KUKA KRL program: EPS_2_251349_CBMH112_A_20251001124303.src

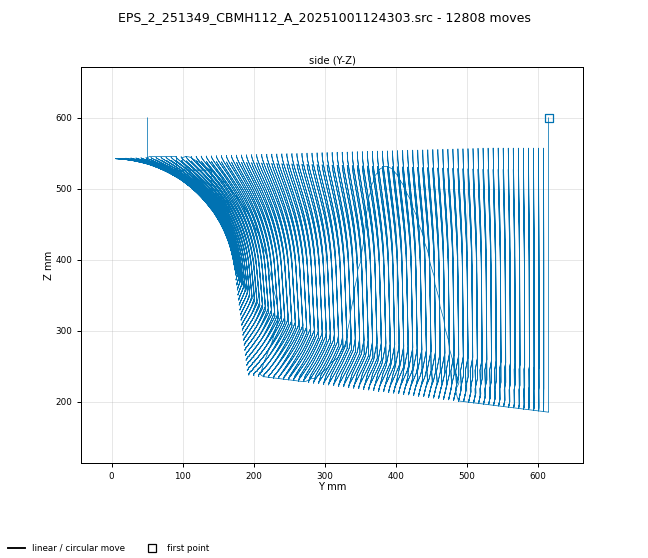
[picture p0: tool path of EPS_2_251349_CBMH112_A_20251001124303.src, 12808 of 12810 moves have a stored position in this frame; points joined in program order, loops and branches not executed]
&ACCESS RVP
&REL 4
&COMMENT QRS 19112012
&PARAM EDITMASK = *
DEF PART()
EXT BAS (BAS_COMMAND :IN,REAL :IN )
INT I
BAS (#INITMOV,0 )

;KUKA QRS Post kuka4.cps  Date:22-06-2017 !

File_ID=2860

QRS_PRE_INIT()

;Init var - Until changes are made in qrs_pre_init
Outlet_Square_prg=0
Inlet_1_Square_prg=0
Inlet_2_Square_prg=0
Inlet_3_Square_prg=0
Inlet_4_Square_prg=0
Inlet_5_Square_prg=0

Outlet_1={X 0.000, Y 529.100, Z 408.000, B 0.000, E1 0.000 }
Inlet_1={X 0.000, Y 531.280, Z 378.000, B 0.000, E1 180.000 }
Outlet_1_type=299
Inlet_1_type=299
;QRS#1=Sidecore dimensions
;QRS#2=300-12" PVC SDR 35
;QRS#3=300-12" PVC SDR 35
;QRS#4=
;QRS#5=
;QRS#6=
;QRS#7=
;QRS#8=
;QRS#9=16M PSX
;QRS#10=16M PSX
;QRS#11=
;QRS#12=
;QRS#13=
;QRS#14=
;QRS#15=
;QRS#16=1220x127x838 2,75'
;QRS#17=EPS Height
;QRS#18=557,5
;QRS#19=*
;QRS#20= UPDATED VERSION 22-06-2017
;QRS#21=*
Outlet_Square=0150
Inlet_1_Square=0150
Inlet_2_Square=0
Inlet_3_Square=0
Inlet_4_Square=0
Inlet_5_Square=0
Mill_Square=1
Outlet_Square_Prg=206
Inlet_1_Square_prg=206

QRS_INIT()

$ADVANCE=5

; T1
PTP {E1 173.597,E2 173.597}
PTP {X 0,Y 615.502,A -85,B 0,C 180,E1 173.597,E2 173.597,E3 0,E4 0,E5 0,E6 0}
QRS_SPEED_INIT()
LIN {X 0,Y 615.502,Z 600,A -85,B 0,C 180,E1 173.597,E2 173.597,E3 0,E4 0,E5 0,E6 0} C_VEL
LIN {X 0,Y 615.502,Z 195.488,A -85,B 0,C 180,E1 173.597,E2 173.597} C_VEL
LIN {X 0,Y 615.502,Z 187.309,A -85,B 0,C 180,E1 173.597,E2 173.597} C_VEL
LIN {X 0,Y 615.487,Z 185.309,A -85,B 0,C 180,E1 173.411,E2 173.411} C_VEL
LIN {X 0,Y 615.496,Z 185.324,A -85,B 0,C 180,E1 170.801,E2 170.801} C_VEL
LIN {X 0,Y 615.474,Z 185.313,A -85,B 0,C 180,E1 168.139,E2 168.139} C_VEL
LIN {X 0,Y 615.483,Z 185.311,A -85,B 0,C 180,E1 165.451,E2 165.451} C_VEL
LIN {X 0,Y 615.488,Z 185.323,A -85,B 0,C 180,E1 162.729,E2 162.729} C_VEL
LIN {X 0,Y 615.489,Z 185.307,A -85,B 0,C 180,E1 159.967,E2 159.967} C_VEL
LIN {X 0,Y 615.483,Z 185.321,A -85,B 0,C 180,E1 157.155,E2 157.155} C_VEL
LIN {X 0,Y 615.476,Z 185.315,A -85,B 0,C 180,E1 154.431,E2 154.431} C_VEL
LIN {X 0,Y 615.483,Z 185.309,A -85,B 0,C 180,E1 152.085,E2 152.085} C_VEL
LIN {X 0,Y 615.488,Z 185.308,A -85,B 0,C 180,E1 149.84,E2 149.84} C_VEL
LIN {X 0,Y 615.477,Z 185.315,A -85,B 0,C 180,E1 147.542,E2 147.542} C_VEL
LIN {X 0,Y 615.491,Z 185.323,A -85,B 0,C 180,E1 145.185,E2 145.185} C_VEL
LIN {X 0,Y 615.479,Z 185.318,A -85,B 0,C 180,E1 142.757,E2 142.757} C_VEL
LIN {X 0,Y 615.483,Z 185.31,A -85,B 0,C 180,E1 139.91,E2 139.91} C_VEL
LIN {X 0,Y 615.477,Z 185.316,A -85,B 0,C 180,E1 137.646,E2 137.646} C_VEL
LIN {X 0,Y 615.482,Z 185.319,A -85,B 0,C 180,E1 134.931,E2 134.931} C_VEL
LIN {X 0,Y 615.484,Z 185.309,A -85,B 0,C 180,E1 132.08,E2 132.08} C_VEL
LIN {X 0,Y 615.476,Z 185.316,A -85,B 0,C 180,E1 129.75,E2 129.75} C_VEL
LIN {X 0,Y 615.48,Z 185.317,A -85,B 0,C 180,E1 126.936,E2 126.936} C_VEL
LIN {X 0,Y 615.483,Z 185.311,A -85,B 0,C 180,E1 124.7,E2 124.7} C_VEL
LIN {X 0,Y 615.489,Z 185.307,A -85,B 0,C 180,E1 122.331,E2 122.331} C_VEL
LIN {X 0,Y 615.491,Z 185.326,A -85,B 0,C 180,E1 119.405,E2 119.405} C_VEL
LIN {X 0,Y 615.485,Z 185.308,A -85,B 0,C 180,E1 116.444,E2 116.444} C_VEL
LIN {X 0,Y 615.485,Z 185.327,A -85,B 0,C 180,E1 113.556,E2 113.556} C_VEL
LIN {X 0,Y 615.476,Z 185.338,A -85,B 0,C 180,E1 112.266,E2 112.266} C_VEL
LIN {X 0,Y 615.46,Z 205.213,A -85,B 0,C 180,E1 109.685,E2 109.685} C_VEL
LIN {X 0,Y 615.464,Z 216.791,A -85,B 0,C 180,E1 108.2,E2 108.2} C_VEL
LIN {X 0,Y 615.491,Z 381.255,A -85,B 0,C 180,E1 106.201,E2 106.201} C_VEL
LIN {X 0,Y 615.489,Z 395.834,A -85,B 0,C 180,E1 105.905,E2 105.905} C_VEL
LIN {X 0,Y 615.477,Z 410.429,A -85,B 0,C 180,E1 105.48,E2 105.48} C_VEL
LIN {X 0,Y 615.492,Z 423.747,A -85,B 0,C 180,E1 104.971,E2 104.971} C_VEL
LIN {X 0,Y 615.483,Z 437.385,A -85,B 0,C 180,E1 104.319,E2 104.319} C_VEL
LIN {X 0,Y 615.5,Z 450.671,A -85,B 0,C 180,E1 103.537,E2 103.537} C_VEL
LIN {X 0,Y 615.497,Z 462.521,A -85,B 0,C 180,E1 102.697,E2 102.697} C_VEL
LIN {X 0,Y 615.497,Z 474.363,A -85,B 0,C 180,E1 101.693,E2 101.693} C_VEL
LIN {X 0,Y 615.495,Z 484.168,A -85,B 0,C 180,E1 100.708,E2 100.708} C_VEL
LIN {X 0,Y 615.495,Z 494.014,A -85,B 0,C 180,E1 99.53,E2 99.53} C_VEL
LIN {X 0,Y 615.496,Z 502.104,A -85,B 0,C 180,E1 98.371,E2 98.371} C_VEL
LIN {X 0,Y 615.491,Z 508.784,A -85,B 0,C 180,E1 97.215,E2 97.215} C_VEL
LIN {X 0,Y 615.499,Z 514.949,A -85,B 0,C 180,E1 95.898,E2 95.898} C_VEL
LIN {X 0,Y 615.489,Z 519.717,A -85,B 0,C 180,E1 94.584,E2 94.584} C_VEL
LIN {X 0,Y 615.491,Z 523.221,A -85,B 0,C 180,E1 93.273,E2 93.273} C_VEL
LIN {X 0,Y 615.5,Z 525.54,A -85,B 0,C 180,E1 91.963,E2 91.963} C_VEL
LIN {X 0,Y 615.491,Z 526.728,A -85,B 0,C 180,E1 90.654,E2 90.654} C_VEL
LIN {X 0,Y 615.492,Z 526.751,A -85,B 0,C 180,E1 89.346,E2 89.346} C_VEL
LIN {X 0,Y 615.5,Z 525.646,A -85,B 0,C 180,E1 88.037,E2 88.037} C_VEL
LIN {X 0,Y 615.494,Z 523.416,A -85,B 0,C 180,E1 86.727,E2 86.727} C_VEL
LIN {X 0,Y 615.49,Z 520.005,A -85,B 0,C 180,E1 85.416,E2 85.416} C_VEL
LIN {X 0,Y 615.499,Z 515.336,A -85,B 0,C 180,E1 84.102,E2 84.102} C_VEL
LIN {X 0,Y 615.49,Z 509.273,A -85,B 0,C 180,E1 82.785,E2 82.785} C_VEL
LIN {X 0,Y 615.493,Z 501.634,A -85,B 0,C 180,E1 81.464,E2 81.464} C_VEL
LIN {X 0,Y 615.496,Z 493.451,A -85,B 0,C 180,E1 80.304,E2 80.304} C_VEL
LIN {X 0,Y 615.495,Z 483.338,A -85,B 0,C 180,E1 79.109,E2 79.109} C_VEL
LIN {X 0,Y 615.497,Z 471.686,A -85,B 0,C 180,E1 77.973,E2 77.973} C_VEL
LIN {X 0,Y 615.498,Z 460.416,A -85,B 0,C 180,E1 77.051,E2 77.051} C_VEL
LIN {X 0,Y 615.498,Z 448.178,A -85,B 0,C 180,E1 76.211,E2 76.211} C_VEL
LIN {X 0,Y 615.484,Z 434.781,A -85,B 0,C 180,E1 75.451,E2 75.451} C_VEL
LIN {X 0,Y 615.488,Z 419.868,A -85,B 0,C 180,E1 74.774,E2 74.774} C_VEL
LIN {X 0,Y 615.476,Z 405.395,A -85,B 0,C 180,E1 74.265,E2 74.265} C_VEL
LIN {X 0,Y 615.492,Z 389.76,A -85,B 0,C 180,E1 73.865,E2 73.865} C_VEL
LIN {X 0,Y 615.492,Z 374.754,A -85,B 0,C 180,E1 73.618,E2 73.618} C_VEL
LIN {X 0,Y 615.471,Z 216.859,A -85,B 0,C 180,E1 71.719,E2 71.719} C_VEL
LIN {X 0,Y 615.478,Z 195.117,A -85,B 0,C 180,E1 68.919,E2 68.919} C_VEL
LIN {X 0,Y 615.483,Z 185.31,A -85,B 0,C 180,E1 67.625,E2 67.625} C_VEL
LIN {X 0,Y 615.478,Z 185.313,A -85,B 0,C 180,E1 65.008,E2 65.008} C_VEL
LIN {X 0,Y 615.476,Z 185.318,A -85,B 0,C 180,E1 62.823,E2 62.823} C_VEL
LIN {X 0,Y 615.482,Z 185.319,A -85,B 0,C 180,E1 60.207,E2 60.207} C_VEL
LIN {X 0,Y 615.493,Z 185.306,A -85,B 0,C 180,E1 57.544,E2 57.544} C_VEL
LIN {X 0,Y 615.478,Z 185.312,A -85,B 0,C 180,E1 55.185,E2 55.185} C_VEL
LIN {X 0,Y 615.486,Z 185.322,A -85,B 0,C 180,E1 52.759,E2 52.759} C_VEL
LIN {X 0,Y 615.482,Z 185.31,A -85,B 0,C 180,E1 49.912,E2 49.912} C_VEL
LIN {X 0,Y 615.495,Z 185.306,A -85,B 0,C 180,E1 47.649,E2 47.649} C_VEL
LIN {X 0,Y 615.479,Z 185.322,A -85,B 0,C 180,E1 44.932,E2 44.932} C_VEL
LIN {X 0,Y 615.483,Z 185.311,A -85,B 0,C 180,E1 42.081,E2 42.081} C_VEL
LIN {X 0,Y 615.489,Z 185.307,A -85,B 0,C 180,E1 39.75,E2 39.75} C_VEL
LIN {X 0,Y 615.482,Z 185.325,A -85,B 0,C 180,E1 36.938,E2 36.938} C_VEL
LIN {X 0,Y 615.488,Z 185.308,A -85,B 0,C 180,E1 34.022,E2 34.022} C_VEL
LIN {X 0,Y 615.479,Z 185.323,A -85,B 0,C 180,E1 31.087,E2 31.087} C_VEL
LIN {X 0,Y 615.481,Z 185.314,A -85,B 0,C 180,E1 28.452,E2 28.452} C_VEL
LIN {X 0,Y 615.476,Z 185.311,A -85,B 0,C 180,E1 25.716,E2 25.716} C_VEL
LIN {X 0,Y 615.473,Z 185.315,A -85,B 0,C 180,E1 23.557,E2 23.557} C_VEL
LIN {X 0,Y 615.475,Z 185.318,A -85,B 0,C 180,E1 21.432,E2 21.432} C_VEL
LIN {X 0,Y 615.482,Z 185.314,A -85,B 0,C 180,E1 18.607,E2 18.607} C_VEL
LIN {X 0,Y 615.477,Z 185.311,A -85,B 0,C 180,E1 15.906,E2 15.906} C_VEL
LIN {X 0,Y 615.492,Z 185.325,A -85,B 0,C 180,E1 13.201,E2 13.201} C_VEL
LIN {X 0,Y 615.488,Z 185.31,A -85,B 0,C 180,E1 10.527,E2 10.527} C_VEL
LIN {X 0,Y 615.471,Z 185.314,A -85,B 0,C 180,E1 7.876,E2 7.876} C_VEL
LIN {X 0,Y 615.495,Z 185.325,A -85,B 0,C 180,E1 5.241,E2 5.241} C_VEL
LIN {X 0,Y 615.49,Z 185.309,A -85,B 0,C 180,E1 2.618,E2 2.618} C_VEL
LIN {X 0,Y 615.47,Z 185.314,A -85,B 0,C 180,E1 0,E2 0} C_VEL
LIN {X 0,Y 615.491,Z 185.327,A -85,B 0,C 180,E1 -2.618,E2 -2.618} C_VEL
LIN {X 0,Y 615.49,Z 185.309,A -85,B 0,C 180,E1 -5.241,E2 -5.241} C_VEL
LIN {X 0,Y 615.469,Z 185.314,A -85,B 0,C 180,E1 -7.876,E2 -7.876} C_VEL
LIN {X 0,Y 615.491,Z 185.327,A -85,B 0,C 180,E1 -10.527,E2 -10.527} C_VEL
LIN {X 0,Y 615.495,Z 185.307,A -85,B 0,C 180,E1 -13.201,E2 -13.201} C_VEL
LIN {X 0,Y 615.468,Z 185.316,A -85,B 0,C 180,E1 -15.906,E2 -15.906} C_VEL
LIN {X 0,Y 615.488,Z 185.319,A -85,B 0,C 180,E1 -18.646,E2 -18.646} C_VEL
LIN {X 0,Y 615.472,Z 185.311,A -85,B 0,C 180,E1 -21.432,E2 -21.432} C_VEL
LIN {X 0,Y 615.487,Z 185.326,A -85,B 0,C 180,E1 -24.272,E2 -24.272} C_VEL
LIN {X 0,Y 615.487,Z 185.308,A -85,B 0,C 180,E1 -27.177,E2 -27.177} C_VEL
LIN {X 0,Y 615.468,Z 185.318,A -85,B 0,C 180,E1 -29.794,E2 -29.794} C_VEL
LIN {X 0,Y 615.488,Z 185.319,A -85,B 0,C 180,E1 -32.457,E2 -32.457} C_VEL
LIN {X 0,Y 615.493,Z 185.309,A -85,B 0,C 180,E1 -34.815,E2 -34.815} C_VEL
LIN {X 0,Y 615.47,Z 185.312,A -85,B 0,C 180,E1 -37.243,E2 -37.243} C_VEL
LIN {X 0,Y 615.495,Z 185.326,A -85,B 0,C 180,E1 -40.091,E2 -40.091} C_VEL
LIN {X 0,Y 615.476,Z 185.31,A -85,B 0,C 180,E1 -43.048,E2 -43.048} C_VEL
LIN {X 0,Y 615.484,Z 185.323,A -85,B 0,C 180,E1 -45.851,E2 -45.851} C_VEL
LIN {X 0,Y 615.492,Z 185.311,A -85,B 0,C 180,E1 -48.528,E2 -48.528} C_VEL
LIN {X 0,Y 615.466,Z 185.313,A -85,B 0,C 180,E1 -51.095,E2 -51.095} C_VEL
LIN {X 0,Y 615.471,Z 185.32,A -85,B 0,C 180,E1 -53.575,E2 -53.575} C_VEL
LIN {X 0,Y 615.495,Z 185.309,A -85,B 0,C 180,E1 -56.465,E2 -56.465} C_VEL
LIN {X 0,Y 615.46,Z 185.315,A -85,B 0,C 180,E1 -59.08,E2 -59.08} C_VEL
LIN {X 0,Y 615.477,Z 185.322,A -85,B 0,C 180,E1 -61.552,E2 -61.552} C_VEL
LIN {X 0,Y 615.498,Z 185.307,A -85,B 0,C 180,E1 -64.429,E2 -64.429} C_VEL
LIN {X 0,Y 615.462,Z 185.437,A -85,B 0,C 180,E1 -64.935,E2 -64.935} C_VEL
LIN {X 0,Y 615.485,Z 209.182,A -85,B 0,C 180,E1 -67.654,E2 -67.654} C_VEL
LIN {X 0,Y 615.495,Z 234.441,A -85,B 0,C 180,E1 -70.489,E2 -70.489} C_VEL
LIN {X 0,Y 615.487,Z 246.053,A -85,B 0,C 180,E1 -71.762,E2 -71.762} C_VEL
LIN {X 0,Y 615.483,Z 412.217,A -85,B 0,C 180,E1 -73.769,E2 -73.769} C_VEL
LIN {X 0,Y 615.496,Z 427.729,A -85,B 0,C 180,E1 -74.095,E2 -74.095} C_VEL
LIN {X 0,Y 615.481,Z 443.062,A -85,B 0,C 180,E1 -74.562,E2 -74.562} C_VEL
LIN {X 0,Y 615.497,Z 456.762,A -85,B 0,C 180,E1 -75.113,E2 -75.113} C_VEL
LIN {X 0,Y 615.495,Z 471.048,A -85,B 0,C 180,E1 -75.834,E2 -75.834} C_VEL
LIN {X 0,Y 615.497,Z 483.904,A -85,B 0,C 180,E1 -76.631,E2 -76.631} C_VEL
LIN {X 0,Y 615.495,Z 496.259,A -85,B 0,C 180,E1 -77.554,E2 -77.554} C_VEL
LIN {X 0,Y 615.495,Z 506.61,A -85,B 0,C 180,E1 -78.474,E2 -78.474} C_VEL
LIN {X 0,Y 615.495,Z 516.186,A -85,B 0,C 180,E1 -79.473,E2 -79.473} C_VEL
LIN {X 0,Y 615.493,Z 525.579,A -85,B 0,C 180,E1 -80.636,E2 -80.636} C_VEL
LIN {X 0,Y 615.494,Z 533.382,A -85,B 0,C 180,E1 -81.794,E2 -81.794} C_VEL
LIN {X 0,Y 615.496,Z 540.606,A -85,B 0,C 180,E1 -83.102,E2 -83.102} C_VEL
LIN {X 0,Y 615.499,Z 546.437,A -85,B 0,C 180,E1 -84.43,E2 -84.43} C_VEL
LIN {X 0,Y 615.491,Z 549.861,A -85,B 0,C 180,E1 -85.416,E2 -85.416} C_VEL
LIN {X 0,Y 615.492,Z 553.318,A -85,B 0,C 180,E1 -86.727,E2 -86.727} C_VEL
LIN {X 0,Y 615.499,Z 555.593,A -85,B 0,C 180,E1 -88.037,E2 -88.037} C_VEL
LIN {X 0,Y 615.493,Z 556.74,A -85,B 0,C 180,E1 -89.346,E2 -89.346} C_VEL
LIN {X 0,Y 615.493,Z 556.74,A -85,B 0,C 180,E1 -90.654,E2 -90.654} C_VEL
LIN {X 0,Y 615.499,Z 555.593,A -85,B 0,C 180,E1 -91.963,E2 -91.963} C_VEL
LIN {X 0,Y 615.492,Z 553.318,A -85,B 0,C 180,E1 -93.273,E2 -93.273} C_VEL
LIN {X 0,Y 615.491,Z 549.86,A -85,B 0,C 180,E1 -94.584,E2 -94.584} C_VEL
LIN {X 0,Y 615.499,Z 545.142,A -85,B 0,C 180,E1 -95.898,E2 -95.898} C_VEL
LIN {X 0,Y 615.494,Z 539.03,A -85,B 0,C 180,E1 -97.215,E2 -97.215} C_VEL
LIN {X 0,Y 615.494,Z 531.334,A -85,B 0,C 180,E1 -98.536,E2 -98.536} C_VEL
LIN {X 0,Y 615.495,Z 523.115,A -85,B 0,C 180,E1 -99.696,E2 -99.696} C_VEL
LIN {X 0,Y 615.497,Z 512.891,A -85,B 0,C 180,E1 -100.893,E2 -100.893} C_VEL
LIN {X 0,Y 615.495,Z 503.07,A -85,B 0,C 180,E1 -101.86,E2 -101.86} C_VEL
LIN {X 0,Y 615.497,Z 490.951,A -85,B 0,C 180,E1 -102.865,E2 -102.865} C_VEL
LIN {X 0,Y 615.498,Z 478.802,A -85,B 0,C 180,E1 -103.705,E2 -103.705} C_VEL
LIN {X 0,Y 615.488,Z 465.384,A -85,B 0,C 180,E1 -104.472,E2 -104.472} C_VEL
LIN {X 0,Y 615.497,Z 450.856,A -85,B 0,C 180,E1 -105.141,E2 -105.141} C_VEL
LIN {X 0,Y 615.495,Z 436.626,A -85,B 0,C 180,E1 -105.65,E2 -105.65} C_VEL
LIN {X 0,Y 615.498,Z 422.155,A -85,B 0,C 180,E1 -106.035,E2 -106.035} C_VEL
LIN {X 0,Y 615.484,Z 407.623,A -85,B 0,C 180,E1 -106.297,E2 -106.297} C_VEL
LIN {X 0,Y 615.489,Z 245.745,A -85,B 0,C 180,E1 -108.258,E2 -108.258} C_VEL
LIN {X 0,Y 615.49,Z 220.396,A -85,B 0,C 180,E1 -111.08,E2 -111.08} C_VEL
LIN {X 0,Y 615.49,Z 194.589,A -85,B 0,C 180,E1 -114.009,E2 -114.009} C_VEL
LIN {X 0,Y 615.463,Z 185.313,A -85,B 0,C 180,E1 -115.101,E2 -115.101} C_VEL
LIN {X 0,Y 615.489,Z 185.317,A -85,B 0,C 180,E1 -117.914,E2 -117.914} C_VEL
LIN {X 0,Y 615.498,Z 185.325,A -85,B 0,C 180,E1 -120.159,E2 -120.159} C_VEL
LIN {X 0,Y 615.473,Z 185.321,A -85,B 0,C 180,E1 -122.458,E2 -122.458} C_VEL
LIN {X 0,Y 615.462,Z 185.315,A -85,B 0,C 180,E1 -124.816,E2 -124.816} C_VEL
LIN {X 0,Y 615.481,Z 185.309,A -85,B 0,C 180,E1 -127.242,E2 -127.242} C_VEL
LIN {X 0,Y 615.496,Z 185.325,A -85,B 0,C 180,E1 -130.09,E2 -130.09} C_VEL
LIN {X 0,Y 615.472,Z 185.32,A -85,B 0,C 180,E1 -132.353,E2 -132.353} C_VEL
LIN {X 0,Y 615.476,Z 185.31,A -85,B 0,C 180,E1 -135.068,E2 -135.068} C_VEL
LIN {X 0,Y 615.493,Z 185.326,A -85,B 0,C 180,E1 -137.918,E2 -137.918} C_VEL
LIN {X 0,Y 615.473,Z 185.32,A -85,B 0,C 180,E1 -140.249,E2 -140.249} C_VEL
LIN {X 0,Y 615.484,Z 185.309,A -85,B 0,C 180,E1 -143.062,E2 -143.062} C_VEL
LIN {X 0,Y 615.486,Z 185.323,A -85,B 0,C 180,E1 -145.978,E2 -145.978} C_VEL
LIN {X 0,Y 615.467,Z 185.317,A -85,B 0,C 180,E1 -148.314,E2 -148.314} C_VEL
LIN {X 0,Y 615.471,Z 185.312,A -85,B 0,C 180,E1 -150.593,E2 -150.593} C_VEL
LIN {X 0,Y 615.497,Z 185.306,A -85,B 0,C 180,E1 -152.951,E2 -152.951} C_VEL
LIN {X 0,Y 615.488,Z 185.327,A -85,B 0,C 180,E1 -155.728,E2 -155.728} C_VEL
LIN {X 0,Y 615.473,Z 185.311,A -85,B 0,C 180,E1 -158.568,E2 -158.568} C_VEL
LIN {X 0,Y 615.487,Z 185.319,A -85,B 0,C 180,E1 -161.391,E2 -161.391} C_VEL
LIN {X 0,Y 615.47,Z 185.317,A -85,B 0,C 180,E1 -164.094,E2 -164.094} C_VEL
LIN {X 0,Y 615.495,Z 185.307,A -85,B 0,C 180,E1 -166.799,E2 -166.799} C_VEL
LIN {X 0,Y 615.493,Z 185.325,A -85,B 0,C 180,E1 -169.473,E2 -169.473} C_VEL
LIN {X 0,Y 615.471,Z 185.314,A -85,B 0,C 180,E1 -172.124,E2 -172.124} C_VEL
LIN {X 0,Y 615.489,Z 185.309,A -85,B 0,C 180,E1 -174.759,E2 -174.759} C_VEL
LIN {X 0,Y 615.494,Z 185.325,A -85,B 0,C 180,E1 -177.382,E2 -177.382} C_VEL
LIN {X 0,Y 615.472,Z 185.314,A -85,B 0,C 180,E1 -180,E2 -180} C_VEL
LIN {X 0,Y 615.489,Z 185.308,A -85,B 0,C 180,E1 -182.618,E2 -182.618} C_VEL
LIN {X 0,Y 615.495,Z 185.324,A -85,B 0,C 180,E1 -185.241,E2 -185.241} C_VEL
LIN {X 0,Y 615.487,Z 185.309,A -85,B 0,C 180,E1 -186.589,E2 -186.589} C_VEL
LIN {X 0,Y 614.813,Z 185.47,A -85,B 0,C 180,E1 -187.135,E2 -187.135} C_VEL
LIN {X 0,Y 611.984,Z 185.873,A -85,B 0,C 180,E1 -188.021,E2 -188.021} C_VEL
LIN {X 0,Y 609.593,Z 186.19,A -85,B 0,C 180,E1 -188.734,E2 -188.734} C_VEL
LIN {X 0,Y 608.552,Z 186.311,A -85,B 0,C 180,E1 -189.283,E2 -189.283} C_VEL
LIN {X 0,Y 608.459,Z 186.318,A -85,B 0,C 180,E1 -189.47,E2 -189.47} C_VEL
LIN {X 0,Y 608.452,Z 186.313,A -85,B 0,C 180,E1 -192,E2 -192} C_VEL
LIN {X 0,Y 608.473,Z 186.313,A -85,B 0,C 180,E1 -194.721,E2 -194.721} C_VEL
LIN {X 0,Y 608.45,Z 186.318,A -85,B 0,C 180,E1 -197.477,E2 -197.477} C_VEL
LIN {X 0,Y 608.46,Z 186.312,A -85,B 0,C 180,E1 -200.274,E2 -200.274} C_VEL
LIN {X 0,Y 608.448,Z 186.315,A -85,B 0,C 180,E1 -202.477,E2 -202.477} C_VEL
LIN {X 0,Y 608.456,Z 186.315,A -85,B 0,C 180,E1 -204.571,E2 -204.571} C_VEL
LIN {X 0,Y 608.48,Z 186.316,A -85,B 0,C 180,E1 -207.21,E2 -207.21} C_VEL
LIN {X 0,Y 608.466,Z 186.311,A -85,B 0,C 180,E1 -209.974,E2 -209.974} C_VEL
LIN {X 0,Y 608.452,Z 186.316,A -85,B 0,C 180,E1 -212.523,E2 -212.523} C_VEL
LIN {X 0,Y 608.442,Z 186.318,A -85,B 0,C 180,E1 -215.278,E2 -215.278} C_VEL
LIN {X 0,Y 608.465,Z 186.311,A -85,B 0,C 180,E1 -217.747,E2 -217.747} C_VEL
LIN {X 0,Y 608.447,Z 186.316,A -85,B 0,C 180,E1 -220.33,E2 -220.33} C_VEL
LIN {X 0,Y 608.448,Z 186.321,A -85,B 0,C 180,E1 -222.96,E2 -222.96} C_VEL
LIN {X 0,Y 608.458,Z 186.312,A -85,B 0,C 180,E1 -225.736,E2 -225.736} C_VEL
LIN {X 0,Y 608.46,Z 186.321,A -85,B 0,C 180,E1 -228.658,E2 -228.658} C_VEL
LIN {X 0,Y 608.462,Z 186.312,A -85,B 0,C 180,E1 -231.413,E2 -231.413} C_VEL
LIN {X 0,Y 608.443,Z 186.315,A -85,B 0,C 180,E1 -233.955,E2 -233.955} C_VEL
LIN {X 0,Y 608.463,Z 186.317,A -85,B 0,C 180,E1 -236.33,E2 -236.33} C_VEL
LIN {X 0,Y 608.459,Z 186.32,A -85,B 0,C 180,E1 -238.731,E2 -238.731} C_VEL
LIN {X 0,Y 608.473,Z 186.31,A -85,B 0,C 180,E1 -241.38,E2 -241.38} C_VEL
LIN {X 0,Y 608.471,Z 186.317,A -85,B 0,C 180,E1 -244.279,E2 -244.279} C_VEL
LIN {X 0,Y 608.449,Z 186.318,A -85,B 0,C 180,E1 -246.877,E2 -246.877} C_VEL
LIN {X 0,Y 608.477,Z 186.333,A -85,B 0,C 180,E1 -247.595,E2 -247.595} C_VEL
LIN {X 0,Y 608.58,Z 202.526,A -85,B 0,C 180,E1 -249.73,E2 -249.73} C_VEL
LIN {X 0,Y 608.525,Z 216.817,A -85,B 0,C 180,E1 -251.585,E2 -251.585} C_VEL
LIN {X 0,Y 608.723,Z 220.642,A -85,B 0,C 180,E1 -251.653,E2 -251.653} C_VEL
LIN {X 0,Y 608.69,Z 382.355,A -85,B 0,C 180,E1 -253.63,E2 -253.63} C_VEL
LIN {X 0,Y 608.647,Z 397.654,A -85,B 0,C 180,E1 -253.955,E2 -253.955} C_VEL
LIN {X 0,Y 608.61,Z 413.004,A -85,B 0,C 180,E1 -254.426,E2 -254.426} C_VEL
LIN {X 0,Y 608.597,Z 427.682,A -85,B 0,C 180,E1 -255.026,E2 -255.026} C_VEL
LIN {X 0,Y 608.57,Z 441.447,A -85,B 0,C 180,E1 -255.735,E2 -255.735} C_VEL
LIN {X 0,Y 608.547,Z 454.549,A -85,B 0,C 180,E1 -256.561,E2 -256.561} C_VEL
LIN {X 0,Y 608.505,Z 466.844,A -85,B 0,C 180,E1 -257.494,E2 -257.494} C_VEL
LIN {X 0,Y 608.497,Z 478.053,A -85,B 0,C 180,E1 -258.508,E2 -258.508} C_VEL
LIN {X 0,Y 608.477,Z 488.937,A -85,B 0,C 180,E1 -259.687,E2 -259.687} C_VEL
LIN {X 0,Y 608.469,Z 497.985,A -85,B 0,C 180,E1 -260.862,E2 -260.862} C_VEL
LIN {X 0,Y 608.457,Z 505.481,A -85,B 0,C 180,E1 -262.033,E2 -262.033} C_VEL
LIN {X 0,Y 608.445,Z 512.63,A -85,B 0,C 180,E1 -263.397,E2 -263.397} C_VEL
LIN {X 0,Y 608.435,Z 517.994,A -85,B 0,C 180,E1 -264.698,E2 -264.698} C_VEL
LIN {X 0,Y 608.432,Z 522.167,A -85,B 0,C 180,E1 -266.026,E2 -266.026} C_VEL
LIN {X 0,Y 608.421,Z 525.11,A -85,B 0,C 180,E1 -267.352,E2 -267.352} C_VEL
LIN {X 0,Y 608.444,Z 526.88,A -85,B 0,C 180,E1 -268.676,E2 -268.676} C_VEL
LIN {X 0,Y 608.432,Z 527.495,A -85,B 0,C 180,E1 -270,E2 -270} C_VEL
LIN {X 0,Y 608.446,Z 526.944,A -85,B 0,C 180,E1 -271.324,E2 -271.324} C_VEL
LIN {X 0,Y 608.424,Z 525.259,A -85,B 0,C 180,E1 -272.648,E2 -272.648} C_VEL
LIN {X 0,Y 608.431,Z 522.408,A -85,B 0,C 180,E1 -273.974,E2 -273.974} C_VEL
LIN {X 0,Y 608.435,Z 518.329,A -85,B 0,C 180,E1 -275.302,E2 -275.302} C_VEL
LIN {X 0,Y 608.445,Z 512.922,A -85,B 0,C 180,E1 -276.633,E2 -276.633} C_VEL
LIN {X 0,Y 608.456,Z 506.024,A -85,B 0,C 180,E1 -277.967,E2 -277.967} C_VEL
LIN {X 0,Y 608.466,Z 498.593,A -85,B 0,C 180,E1 -279.138,E2 -279.138} C_VEL
LIN {X 0,Y 608.476,Z 489.665,A -85,B 0,C 180,E1 -280.313,E2 -280.313} C_VEL
LIN {X 0,Y 608.495,Z 478.949,A -85,B 0,C 180,E1 -281.492,E2 -281.492} C_VEL
LIN {X 0,Y 608.513,Z 466.909,A -85,B 0,C 180,E1 -282.591,E2 -282.591} C_VEL
LIN {X 0,Y 608.543,Z 454.622,A -85,B 0,C 180,E1 -283.524,E2 -283.524} C_VEL
LIN {X 0,Y 608.585,Z 441.681,A -85,B 0,C 180,E1 -284.341,E2 -284.341} C_VEL
LIN {X 0,Y 608.606,Z 427.777,A -85,B 0,C 180,E1 -285.059,E2 -285.059} C_VEL
LIN {X 0,Y 608.627,Z 413.116,A -85,B 0,C 180,E1 -285.659,E2 -285.659} C_VEL
LIN {X 0,Y 608.663,Z 397.536,A -85,B 0,C 180,E1 -286.138,E2 -286.138} C_VEL
LIN {X 0,Y 608.692,Z 382.189,A -85,B 0,C 180,E1 -286.463,E2 -286.463} C_VEL
LIN {X 0,Y 608.7,Z 217.921,A -85,B 0,C 180,E1 -288.471,E2 -288.471} C_VEL
LIN {X 0,Y 608.528,Z 216.877,A -85,B 0,C 180,E1 -288.497,E2 -288.497} C_VEL
LIN {X 0,Y 608.558,Z 196.464,A -85,B 0,C 180,E1 -291.155,E2 -291.155} C_VEL
LIN {X 0,Y 608.471,Z 186.312,A -85,B 0,C 180,E1 -292.506,E2 -292.506} C_VEL
LIN {X 0,Y 608.452,Z 186.319,A -85,B 0,C 180,E1 -295.3,E2 -295.3} C_VEL
LIN {X 0,Y 608.443,Z 186.324,A -85,B 0,C 180,E1 -297.518,E2 -297.518} C_VEL
LIN {X 0,Y 608.462,Z 186.314,A -85,B 0,C 180,E1 -299.97,E2 -299.97} C_VEL
LIN {X 0,Y 608.459,Z 186.314,A -85,B 0,C 180,E1 -302.879,E2 -302.879} C_VEL
LIN {X 0,Y 608.441,Z 186.322,A -85,B 0,C 180,E1 -305.277,E2 -305.277} C_VEL
LIN {X 0,Y 608.466,Z 186.316,A -85,B 0,C 180,E1 -307.745,E2 -307.745} C_VEL
LIN {X 0,Y 608.447,Z 186.313,A -85,B 0,C 180,E1 -310.328,E2 -310.328} C_VEL
LIN {X 0,Y 608.476,Z 186.32,A -85,B 0,C 180,E1 -313.309,E2 -313.309} C_VEL
LIN {X 0,Y 608.468,Z 186.311,A -85,B 0,C 180,E1 -316.13,E2 -316.13} C_VEL
LIN {X 0,Y 608.447,Z 186.317,A -85,B 0,C 180,E1 -318.823,E2 -318.823} C_VEL
LIN {X 0,Y 608.467,Z 186.317,A -85,B 0,C 180,E1 -321.412,E2 -321.412} C_VEL
LIN {X 0,Y 608.474,Z 186.31,A -85,B 0,C 180,E1 -323.949,E2 -323.949} C_VEL
LIN {X 0,Y 608.457,Z 186.312,A -85,B 0,C 180,E1 -326.329,E2 -326.329} C_VEL
LIN {X 0,Y 608.47,Z 186.314,A -85,B 0,C 180,E1 -328.727,E2 -328.727} C_VEL
LIN {X 0,Y 608.469,Z 186.316,A -85,B 0,C 180,E1 -331.378,E2 -331.378} C_VEL
LIN {X 0,Y 608.438,Z 186.314,A -85,B 0,C 180,E1 -333.964,E2 -333.964} C_VEL
LIN {X 0,Y 608.466,Z 186.311,A -85,B 0,C 180,E1 -336.155,E2 -336.155} C_VEL
LIN {X 0,Y 608.449,Z 186.323,A -85,B 0,C 180,E1 -339.018,E2 -339.018} C_VEL
LIN {X 0,Y 608.444,Z 186.313,A -85,B 0,C 180,E1 -341.828,E2 -341.828} C_VEL
LIN {X 0,Y 608.471,Z 186.316,A -85,B 0,C 180,E1 -344.594,E2 -344.594} C_VEL
LIN {X 0,Y 608.476,Z 186.312,A -85,B 0,C 180,E1 -347.323,E2 -347.323} C_VEL
LIN {X 0,Y 608.445,Z 186.314,A -85,B 0,C 180,E1 -350.022,E2 -350.022} C_VEL
LIN {X 0,Y 608.477,Z 186.319,A -85,B 0,C 180,E1 -352.701,E2 -352.701} C_VEL
LIN {X 0,Y 608.457,Z 186.313,A -85,B 0,C 180,E1 -355.362,E2 -355.362} C_VEL
LIN {X 0,Y 608.441,Z 186.315,A -85,B 0,C 180,E1 -358.014,E2 -358.014} C_VEL
LIN {X 0,Y 608.481,Z 186.32,A -85,B 0,C 180,E1 -360.662,E2 -360.662} C_VEL
LIN {X 0,Y 608.478,Z 186.31,A -85,B 0,C 180,E1 -363.311,E2 -363.311} C_VEL
LIN {X 0,Y 608.446,Z 186.315,A -85,B 0,C 180,E1 -365.967,E2 -365.967} C_VEL
LIN {X 0,Y 608.458,Z 186.321,A -85,B 0,C 180,E1 -368.636,E2 -368.636} C_VEL
LIN {X 0,Y 608.471,Z 186.31,A -85,B 0,C 180,E1 -371.324,E2 -371.324} C_VEL
LIN {X 0,Y 608.457,Z 186.315,A -85,B 0,C 180,E1 -374.038,E2 -374.038} C_VEL
LIN {X 0,Y 608.473,Z 186.314,A -85,B 0,C 180,E1 -376.783,E2 -376.783} C_VEL
LIN {X 0,Y 608.446,Z 186.314,A -85,B 0,C 180,E1 -379.571,E2 -379.571} C_VEL
LIN {X 0,Y 608.469,Z 186.319,A -85,B 0,C 180,E1 -382.482,E2 -382.482} C_VEL
LIN {X 0,Y 608.442,Z 186.313,A -85,B 0,C 180,E1 -385.301,E2 -385.301} C_VEL
LIN {X 0,Y 608.443,Z 186.314,A -85,B 0,C 180,E1 -387.518,E2 -387.518} C_VEL
LIN {X 0,Y 608.457,Z 186.318,A -85,B 0,C 180,E1 -389.972,E2 -389.972} C_VEL
LIN {X 0,Y 608.461,Z 186.316,A -85,B 0,C 180,E1 -392.524,E2 -392.524} C_VEL
LIN {X 0,Y 608.434,Z 186.315,A -85,B 0,C 180,E1 -395.278,E2 -395.278} C_VEL
LIN {X 0,Y 608.463,Z 186.315,A -85,B 0,C 180,E1 -397.747,E2 -397.747} C_VEL
LIN {X 0,Y 608.475,Z 186.316,A -85,B 0,C 180,E1 -400.333,E2 -400.333} C_VEL
LIN {X 0,Y 608.445,Z 186.313,A -85,B 0,C 180,E1 -402.96,E2 -402.96} C_VEL
LIN {X 0,Y 608.452,Z 186.318,A -85,B 0,C 180,E1 -405.737,E2 -405.737} C_VEL
LIN {X 0,Y 608.467,Z 186.321,A -85,B 0,C 180,E1 -407.94,E2 -407.94} C_VEL
LIN {X 0,Y 608.468,Z 186.311,A -85,B 0,C 180,E1 -410.703,E2 -410.703} C_VEL
LIN {X 0,Y 608.437,Z 186.315,A -85,B 0,C 180,E1 -413.085,E2 -413.085} C_VEL
LIN {X 0,Y 608.457,Z 186.317,A -85,B 0,C 180,E1 -415.531,E2 -415.531} C_VEL
LIN {X 0,Y 608.466,Z 186.321,A -85,B 0,C 180,E1 -417.906,E2 -417.906} C_VEL
LIN {X 0,Y 608.471,Z 186.314,A -85,B 0,C 180,E1 -420.221,E2 -420.221} C_VEL
LIN {X 0,Y 608.464,Z 186.311,A -85,B 0,C 180,E1 -422.795,E2 -422.795} C_VEL
LIN {X 0,Y 608.473,Z 186.453,A -85,B 0,C 180,E1 -424.746,E2 -424.746} C_VEL
LIN {X 0,Y 608.664,Z 198.547,A -85,B 0,C 180,E1 -426.164,E2 -426.164} C_VEL
LIN {X 0,Y 608.595,Z 221.957,A -85,B 0,C 180,E1 -428.847,E2 -428.847} C_VEL
LIN {X 0,Y 608.574,Z 246.053,A -85,B 0,C 180,E1 -431.547,E2 -431.547} C_VEL
LIN {X 0,Y 608.709,Z 355.316,A -85,B 0,C 180,E1 -432.878,E2 -432.878} C_VEL
LIN {X 0,Y 608.678,Z 412.217,A -85,B 0,C 180,E1 -433.582,E2 -433.582} C_VEL
LIN {X 0,Y 608.671,Z 427.727,A -85,B 0,C 180,E1 -433.912,E2 -433.912} C_VEL
LIN {X 0,Y 608.629,Z 443.06,A -85,B 0,C 180,E1 -434.384,E2 -434.384} C_VEL
LIN {X 0,Y 608.606,Z 456.765,A -85,B 0,C 180,E1 -434.941,E2 -434.941} C_VEL
LIN {X 0,Y 608.578,Z 470.243,A -85,B 0,C 180,E1 -435.625,E2 -435.625} C_VEL
LIN {X 0,Y 608.554,Z 482.669,A -85,B 0,C 180,E1 -436.391,E2 -436.391} C_VEL
LIN {X 0,Y 608.528,Z 495.287,A -85,B 0,C 180,E1 -437.324,E2 -437.324} C_VEL
LIN {X 0,Y 608.496,Z 506.751,A -85,B 0,C 180,E1 -438.339,E2 -438.339} C_VEL
LIN {X 0,Y 608.477,Z 516.391,A -85,B 0,C 180,E1 -439.351,E2 -439.351} C_VEL
LIN {X 0,Y 608.476,Z 525.855,A -85,B 0,C 180,E1 -440.527,E2 -440.527} C_VEL
LIN {X 0,Y 608.456,Z 533.731,A -85,B 0,C 180,E1 -441.699,E2 -441.699} C_VEL
LIN {X 0,Y 608.441,Z 541.088,A -85,B 0,C 180,E1 -443.034,E2 -443.034} C_VEL
LIN {X 0,Y 608.45,Z 546.924,A -85,B 0,C 180,E1 -444.366,E2 -444.366} C_VEL
LIN {X 0,Y 608.427,Z 550.383,A -85,B 0,C 180,E1 -445.362,E2 -445.362} C_VEL
LIN {X 0,Y 608.421,Z 553.886,A -85,B 0,C 180,E1 -446.689,E2 -446.689} C_VEL
LIN {X 0,Y 608.444,Z 556.191,A -85,B 0,C 180,E1 -448.014,E2 -448.014} C_VEL
LIN {X 0,Y 608.436,Z 557.351,A -85,B 0,C 180,E1 -449.338,E2 -449.338} C_VEL
LIN {X 0,Y 608.436,Z 557.351,A -85,B 0,C 180,E1 -450.662,E2 -450.662} C_VEL
LIN {X 0,Y 608.444,Z 556.191,A -85,B 0,C 180,E1 -451.986,E2 -451.986} C_VEL
LIN {X 0,Y 608.421,Z 553.886,A -85,B 0,C 180,E1 -453.311,E2 -453.311} C_VEL
LIN {X 0,Y 608.427,Z 550.383,A -85,B 0,C 180,E1 -454.638,E2 -454.638} C_VEL
LIN {X 0,Y 608.437,Z 545.608,A -85,B 0,C 180,E1 -455.967,E2 -455.967} C_VEL
LIN {X 0,Y 608.457,Z 539.427,A -85,B 0,C 180,E1 -457.299,E2 -457.299} C_VEL
LIN {X 0,Y 608.468,Z 531.655,A -85,B 0,C 180,E1 -458.636,E2 -458.636} C_VEL
LIN {X 0,Y 608.471,Z 523.372,A -85,B 0,C 180,E1 -459.809,E2 -459.809} C_VEL
LIN {X 0,Y 608.492,Z 512.649,A -85,B 0,C 180,E1 -461.063,E2 -461.063} C_VEL
LIN {X 0,Y 608.522,Z 501.278,A -85,B 0,C 180,E1 -462.167,E2 -462.167} C_VEL
LIN {X 0,Y 608.547,Z 489.858,A -85,B 0,C 180,E1 -463.099,E2 -463.099} C_VEL
LIN {X 0,Y 608.562,Z 477.452,A -85,B 0,C 180,E1 -463.95,E2 -463.95} C_VEL
LIN {X 0,Y 608.575,Z 463.866,A -85,B 0,C 180,E1 -464.718,E2 -464.718} C_VEL
LIN {X 0,Y 608.638,Z 449.801,A -85,B 0,C 180,E1 -465.358,E2 -465.358} C_VEL
LIN {X 0,Y 608.645,Z 435.313,A -85,B 0,C 180,E1 -465.873,E2 -465.873} C_VEL
LIN {X 0,Y 608.686,Z 420.036,A -85,B 0,C 180,E1 -466.269,E2 -466.269} C_VEL
LIN {X 0,Y 608.684,Z 404.116,A -85,B 0,C 180,E1 -466.534,E2 -466.534} C_VEL
LIN {X 0,Y 608.683,Z 246.681,A -85,B 0,C 180,E1 -468.441,E2 -468.441} C_VEL
LIN {X 0,Y 608.541,Z 245.57,A -85,B 0,C 180,E1 -468.494,E2 -468.494} C_VEL
LIN {X 0,Y 608.595,Z 221.957,A -85,B 0,C 180,E1 -471.153,E2 -471.153} C_VEL
LIN {X 0,Y 608.664,Z 198.547,A -85,B 0,C 180,E1 -473.836,E2 -473.836} C_VEL
LIN {X 0,Y 608.473,Z 186.452,A -85,B 0,C 180,E1 -475.254,E2 -475.254} C_VEL
LIN {X 0,Y 608.442,Z 186.315,A -85,B 0,C 180,E1 -477.518,E2 -477.518} C_VEL
LIN {X 0,Y 608.47,Z 186.317,A -85,B 0,C 180,E1 -479.972,E2 -479.972} C_VEL
LIN {X 0,Y 608.449,Z 186.313,A -85,B 0,C 180,E1 -482.879,E2 -482.879} C_VEL
LIN {X 0,Y 608.436,Z 186.315,A -85,B 0,C 180,E1 -485.277,E2 -485.277} C_VEL
LIN {X 0,Y 608.466,Z 186.319,A -85,B 0,C 180,E1 -488.24,E2 -488.24} C_VEL
LIN {X 0,Y 608.446,Z 186.319,A -85,B 0,C 180,E1 -490.328,E2 -490.328} C_VEL
LIN {X 0,Y 608.444,Z 186.313,A -85,B 0,C 180,E1 -492.959,E2 -492.959} C_VEL
LIN {X 0,Y 608.459,Z 186.318,A -85,B 0,C 180,E1 -495.734,E2 -495.734} C_VEL
LIN {X 0,Y 608.446,Z 186.314,A -85,B 0,C 180,E1 -498.658,E2 -498.658} C_VEL
LIN {X 0,Y 608.47,Z 186.313,A -85,B 0,C 180,E1 -501.412,E2 -501.412} C_VEL
LIN {X 0,Y 608.468,Z 186.32,A -85,B 0,C 180,E1 -503.95,E2 -503.95} C_VEL
LIN {X 0,Y 608.439,Z 186.317,A -85,B 0,C 180,E1 -506.328,E2 -506.328} C_VEL
LIN {X 0,Y 608.468,Z 186.31,A -85,B 0,C 180,E1 -508.727,E2 -508.727} C_VEL
LIN {X 0,Y 608.472,Z 186.314,A -85,B 0,C 180,E1 -511.378,E2 -511.378} C_VEL
LIN {X 0,Y 608.435,Z 186.321,A -85,B 0,C 180,E1 -513.964,E2 -513.964} C_VEL
LIN {X 0,Y 608.454,Z 186.315,A -85,B 0,C 180,E1 -516.155,E2 -516.155} C_VEL
LIN {X 0,Y 608.459,Z 186.313,A -85,B 0,C 180,E1 -518.308,E2 -518.308} C_VEL
LIN {X 0,Y 608.467,Z 186.315,A -85,B 0,C 180,E1 -521.281,E2 -521.281} C_VEL
LIN {X 0,Y 608.452,Z 186.318,A -85,B 0,C 180,E1 -523.906,E2 -523.906} C_VEL
LIN {X 0,Y 608.465,Z 186.311,A -85,B 0,C 180,E1 -526.644,E2 -526.644} C_VEL
LIN {X 0,Y 608.467,Z 186.318,A -85,B 0,C 180,E1 -529.35,E2 -529.35} C_VEL
LIN {X 0,Y 608.465,Z 186.313,A -85,B 0,C 180,E1 -532.033,E2 -532.033} C_VEL
LIN {X 0,Y 608.466,Z 186.311,A -85,B 0,C 180,E1 -534.698,E2 -534.698} C_VEL
LIN {X 0,Y 608.483,Z 186.318,A -85,B 0,C 180,E1 -537.352,E2 -537.352} C_VEL
LIN {X 0,Y 608.463,Z 186.312,A -85,B 0,C 180,E1 -540,E2 -540} C_VEL
LIN {X 0,Y 608.479,Z 186.31,A -85,B 0,C 180,E1 -542.648,E2 -542.648} C_VEL
LIN {X 0,Y 608.471,Z 186.321,A -85,B 0,C 180,E1 -545.302,E2 -545.302} C_VEL
LIN {X 0,Y 608.467,Z 186.311,A -85,B 0,C 180,E1 -547.967,E2 -547.967} C_VEL
LIN {X 0,Y 608.459,Z 186.318,A -85,B 0,C 180,E1 -549.47,E2 -549.47} C_VEL
LIN {X 0,Y 607.77,Z 186.4,A -85,B 0,C 180,E1 -550.022,E2 -550.022} C_VEL
LIN {X 0,Y 604.91,Z 186.759,A -85,B 0,C 180,E1 -550.919,E2 -550.919} C_VEL
LIN {X 0,Y 602.51,Z 187.056,A -85,B 0,C 180,E1 -551.641,E2 -551.641} C_VEL
LIN {X 0,Y 601.485,Z 187.18,A -85,B 0,C 180,E1 -552.197,E2 -552.197} C_VEL
LIN {X 0,Y 601.404,Z 187.19,A -85,B 0,C 180,E1 -552.386,E2 -552.386} C_VEL
LIN {X 0,Y 601.427,Z 187.193,A -85,B 0,C 180,E1 -554.897,E2 -554.897} C_VEL
LIN {X 0,Y 601.426,Z 187.195,A -85,B 0,C 180,E1 -556.986,E2 -556.986} C_VEL
LIN {X 0,Y 601.404,Z 187.191,A -85,B 0,C 180,E1 -559.81,E2 -559.81} C_VEL
LIN {X 0,Y 601.403,Z 187.195,A -85,B 0,C 180,E1 -562.683,E2 -562.683} C_VEL
LIN {X 0,Y 601.402,Z 187.198,A -85,B 0,C 180,E1 -564.879,E2 -564.879} C_VEL
LIN {X 0,Y 601.417,Z 187.189,A -85,B 0,C 180,E1 -567.868,E2 -567.868} C_VEL
LIN {X 0,Y 601.441,Z 187.186,A -85,B 0,C 180,E1 -570.163,E2 -570.163} C_VEL
LIN {X 0,Y 601.414,Z 187.196,A -85,B 0,C 180,E1 -572.716,E2 -572.716} C_VEL
LIN {X 0,Y 601.411,Z 187.197,A -85,B 0,C 180,E1 -575.116,E2 -575.116} C_VEL
LIN {X 0,Y 601.429,Z 187.189,A -85,B 0,C 180,E1 -577.42,E2 -577.42} C_VEL
LIN {X 0,Y 601.407,Z 187.19,A -85,B 0,C 180,E1 -579.996,E2 -579.996} C_VEL
LIN {X 0,Y 601.406,Z 187.198,A -85,B 0,C 180,E1 -582.671,E2 -582.671} C_VEL
LIN {X 0,Y 601.421,Z 187.189,A -85,B 0,C 180,E1 -585.483,E2 -585.483} C_VEL
LIN {X 0,Y 601.422,Z 187.193,A -85,B 0,C 180,E1 -588.407,E2 -588.407} C_VEL
LIN {X 0,Y 601.428,Z 187.188,A -85,B 0,C 180,E1 -591.53,E2 -591.53} C_VEL
LIN {X 0,Y 601.384,Z 187.197,A -85,B 0,C 180,E1 -594.246,E2 -594.246} C_VEL
LIN {X 0,Y 601.428,Z 187.197,A -85,B 0,C 180,E1 -596.687,E2 -596.687} C_VEL
LIN {X 0,Y 601.418,Z 187.192,A -85,B 0,C 180,E1 -599.059,E2 -599.059} C_VEL
LIN {X 0,Y 601.433,Z 187.188,A -85,B 0,C 180,E1 -601.374,E2 -601.374} C_VEL
LIN {X 0,Y 601.401,Z 187.191,A -85,B 0,C 180,E1 -603.637,E2 -603.637} C_VEL
LIN {X 0,Y 601.417,Z 187.199,A -85,B 0,C 180,E1 -606.59,E2 -606.59} C_VEL
LIN {X 0,Y 601.409,Z 187.199,A -85,B 0,C 180,E1 -607.433,E2 -607.433} C_VEL
LIN {X 0,Y 601.663,Z 191.735,A -85,B 0,C 180,E1 -608.051,E2 -608.051} C_VEL
LIN {X 0,Y 601.602,Z 211.976,A -85,B 0,C 180,E1 -610.73,E2 -610.73} C_VEL
LIN {X 0,Y 601.58,Z 216.857,A -85,B 0,C 180,E1 -611.37,E2 -611.37} C_VEL
LIN {X 0,Y 601.985,Z 220.859,A -85,B 0,C 180,E1 -611.442,E2 -611.442} C_VEL
LIN {X 0,Y 601.888,Z 381.838,A -85,B 0,C 180,E1 -613.43,E2 -613.43} C_VEL
LIN {X 0,Y 601.827,Z 397.675,A -85,B 0,C 180,E1 -613.768,E2 -613.768} C_VEL
LIN {X 0,Y 601.753,Z 413.018,A -85,B 0,C 180,E1 -614.244,E2 -614.244} C_VEL
LIN {X 0,Y 601.725,Z 427.692,A -85,B 0,C 180,E1 -614.851,E2 -614.851} C_VEL
LIN {X 0,Y 601.66,Z 440.99,A -85,B 0,C 180,E1 -615.542,E2 -615.542} C_VEL
LIN {X 0,Y 601.604,Z 453.806,A -85,B 0,C 180,E1 -616.352,E2 -616.352} C_VEL
LIN {X 0,Y 601.541,Z 465.793,A -85,B 0,C 180,E1 -617.261,E2 -617.261} C_VEL
LIN {X 0,Y 601.488,Z 476.283,A -85,B 0,C 180,E1 -618.201,E2 -618.201} C_VEL
LIN {X 0,Y 601.43,Z 485.998,A -85,B 0,C 180,E1 -619.224,E2 -619.224} C_VEL
LIN {X 0,Y 601.428,Z 495.528,A -85,B 0,C 180,E1 -620.415,E2 -620.415} C_VEL
LIN {X 0,Y 601.378,Z 503.461,A -85,B 0,C 180,E1 -621.6,E2 -621.6} C_VEL
LIN {X 0,Y 601.368,Z 510.873,A -85,B 0,C 180,E1 -622.952,E2 -622.952} C_VEL
LIN {X 0,Y 601.373,Z 516.759,A -85,B 0,C 180,E1 -624.299,E2 -624.299} C_VEL
LIN {X 0,Y 601.328,Z 520.242,A -85,B 0,C 180,E1 -625.307,E2 -625.307} C_VEL
LIN {X 0,Y 601.336,Z 523.79,A -85,B 0,C 180,E1 -626.65,E2 -626.65} C_VEL
LIN {X 0,Y 601.343,Z 526.139,A -85,B 0,C 180,E1 -627.991,E2 -627.991} C_VEL
LIN {X 0,Y 601.334,Z 527.337,A -85,B 0,C 180,E1 -629.33,E2 -629.33} C_VEL
LIN {X 0,Y 601.335,Z 527.361,A -85,B 0,C 180,E1 -630.67,E2 -630.67} C_VEL
LIN {X 0,Y 601.343,Z 526.245,A -85,B 0,C 180,E1 -632.009,E2 -632.009} C_VEL
LIN {X 0,Y 601.339,Z 523.983,A -85,B 0,C 180,E1 -633.35,E2 -633.35} C_VEL
LIN {X 0,Y 601.328,Z 520.526,A -85,B 0,C 180,E1 -634.693,E2 -634.693} C_VEL
LIN {X 0,Y 601.358,Z 515.798,A -85,B 0,C 180,E1 -636.037,E2 -636.037} C_VEL
LIN {X 0,Y 601.365,Z 509.667,A -85,B 0,C 180,E1 -637.386,E2 -637.386} C_VEL
LIN {X 0,Y 601.389,Z 501.952,A -85,B 0,C 180,E1 -638.738,E2 -638.738} C_VEL
LIN {X 0,Y 601.428,Z 493.709,A -85,B 0,C 180,E1 -639.925,E2 -639.925} C_VEL
LIN {X 0,Y 601.443,Z 483.367,A -85,B 0,C 180,E1 -641.164,E2 -641.164} C_VEL
LIN {X 0,Y 601.503,Z 471.788,A -85,B 0,C 180,E1 -642.312,E2 -642.312} C_VEL
LIN {X 0,Y 601.557,Z 460.467,A -85,B 0,C 180,E1 -643.254,E2 -643.254} C_VEL
LIN {X 0,Y 601.623,Z 447.319,A -85,B 0,C 180,E1 -644.167,E2 -644.167} C_VEL
LIN {X 0,Y 601.678,Z 434.765,A -85,B 0,C 180,E1 -644.89,E2 -644.89} C_VEL
LIN {X 0,Y 601.756,Z 419.844,A -85,B 0,C 180,E1 -645.582,E2 -645.582} C_VEL
LIN {X 0,Y 601.808,Z 405.357,A -85,B 0,C 180,E1 -646.102,E2 -646.102} C_VEL
LIN {X 0,Y 601.856,Z 389.98,A -85,B 0,C 180,E1 -646.505,E2 -646.505} C_VEL
LIN {X 0,Y 601.898,Z 374.082,A -85,B 0,C 180,E1 -646.771,E2 -646.771} C_VEL
LIN {X 0,Y 601.912,Z 218.646,A -85,B 0,C 180,E1 -648.677,E2 -648.677} C_VEL
LIN {X 0,Y 601.577,Z 216.802,A -85,B 0,C 180,E1 -648.728,E2 -648.728} C_VEL
LIN {X 0,Y 601.669,Z 195.109,A -85,B 0,C 180,E1 -651.588,E2 -651.588} C_VEL
LIN {X 0,Y 601.45,Z 187.238,A -85,B 0,C 180,E1 -652.65,E2 -652.65} C_VEL
LIN {X 0,Y 601.401,Z 187.193,A -85,B 0,C 180,E1 -654.878,E2 -654.878} C_VEL
LIN {X 0,Y 601.41,Z 187.198,A -85,B 0,C 180,E1 -657.361,E2 -657.361} C_VEL
LIN {X 0,Y 601.426,Z 187.189,A -85,B 0,C 180,E1 -660.148,E2 -660.148} C_VEL
LIN {X 0,Y 601.425,Z 187.189,A -85,B 0,C 180,E1 -662.716,E2 -662.716} C_VEL
LIN {X 0,Y 601.406,Z 187.195,A -85,B 0,C 180,E1 -665.113,E2 -665.113} C_VEL
LIN {X 0,Y 601.432,Z 187.198,A -85,B 0,C 180,E1 -667.418,E2 -667.418} C_VEL
LIN {X 0,Y 601.406,Z 187.192,A -85,B 0,C 180,E1 -669.994,E2 -669.994} C_VEL
LIN {X 0,Y 601.41,Z 187.191,A -85,B 0,C 180,E1 -672.669,E2 -672.669} C_VEL
LIN {X 0,Y 601.421,Z 187.196,A -85,B 0,C 180,E1 -675.481,E2 -675.481} C_VEL
LIN {X 0,Y 601.419,Z 187.189,A -85,B 0,C 180,E1 -678.406,E2 -678.406} C_VEL
LIN {X 0,Y 601.431,Z 187.192,A -85,B 0,C 180,E1 -680.875,E2 -680.875} C_VEL
LIN {X 0,Y 601.439,Z 187.188,A -85,B 0,C 180,E1 -683.733,E2 -683.733} C_VEL
LIN {X 0,Y 601.427,Z 187.188,A -85,B 0,C 180,E1 -686.063,E2 -686.063} C_VEL
LIN {X 0,Y 601.434,Z 187.188,A -85,B 0,C 180,E1 -688.541,E2 -688.541} C_VEL
LIN {X 0,Y 601.429,Z 187.193,A -85,B 0,C 180,E1 -691.373,E2 -691.373} C_VEL
LIN {X 0,Y 601.398,Z 187.193,A -85,B 0,C 180,E1 -693.636,E2 -693.636} C_VEL
LIN {X 0,Y 601.416,Z 187.193,A -85,B 0,C 180,E1 -696.589,E2 -696.589} C_VEL
LIN {X 0,Y 601.427,Z 187.19,A -85,B 0,C 180,E1 -699.478,E2 -699.478} C_VEL
LIN {X 0,Y 601.393,Z 187.193,A -85,B 0,C 180,E1 -702.311,E2 -702.311} C_VEL
LIN {X 0,Y 601.413,Z 187.192,A -85,B 0,C 180,E1 -704.409,E2 -704.409} C_VEL
LIN {X 0,Y 601.421,Z 187.193,A -85,B 0,C 180,E1 -707.172,E2 -707.172} C_VEL
LIN {X 0,Y 601.424,Z 187.188,A -85,B 0,C 180,E1 -709.905,E2 -709.905} C_VEL
LIN {X 0,Y 601.446,Z 187.193,A -85,B 0,C 180,E1 -712.615,E2 -712.615} C_VEL
LIN {X 0,Y 601.425,Z 187.19,A -85,B 0,C 180,E1 -715.308,E2 -715.308} C_VEL
LIN {X 0,Y 601.412,Z 187.19,A -85,B 0,C 180,E1 -717.991,E2 -717.991} C_VEL
LIN {X 0,Y 601.451,Z 187.195,A -85,B 0,C 180,E1 -720.669,E2 -720.669} C_VEL
LIN {X 0,Y 601.428,Z 187.188,A -85,B 0,C 180,E1 -723.349,E2 -723.349} C_VEL
LIN {X 0,Y 601.399,Z 187.193,A -85,B 0,C 180,E1 -726.037,E2 -726.037} C_VEL
LIN {X 0,Y 601.437,Z 187.193,A -85,B 0,C 180,E1 -728.738,E2 -728.738} C_VEL
LIN {X 0,Y 601.427,Z 187.188,A -85,B 0,C 180,E1 -731.458,E2 -731.458} C_VEL
LIN {X 0,Y 601.41,Z 187.196,A -85,B 0,C 180,E1 -734.206,E2 -734.206} C_VEL
LIN {X 0,Y 601.428,Z 187.189,A -85,B 0,C 180,E1 -736.986,E2 -736.986} C_VEL
LIN {X 0,Y 601.4,Z 187.193,A -85,B 0,C 180,E1 -739.81,E2 -739.81} C_VEL
LIN {X 0,Y 601.415,Z 187.195,A -85,B 0,C 180,E1 -742.608,E2 -742.608} C_VEL
LIN {X 0,Y 601.399,Z 187.193,A -85,B 0,C 180,E1 -744.879,E2 -744.879} C_VEL
LIN {X 0,Y 601.415,Z 187.193,A -85,B 0,C 180,E1 -747.868,E2 -747.868} C_VEL
LIN {X 0,Y 601.44,Z 187.196,A -85,B 0,C 180,E1 -750.163,E2 -750.163} C_VEL
LIN {X 0,Y 601.419,Z 187.191,A -85,B 0,C 180,E1 -752.717,E2 -752.717} C_VEL
LIN {X 0,Y 601.407,Z 187.19,A -85,B 0,C 180,E1 -755.115,E2 -755.115} C_VEL
LIN {X 0,Y 601.427,Z 187.188,A -85,B 0,C 180,E1 -757.42,E2 -757.42} C_VEL
LIN {X 0,Y 601.401,Z 187.199,A -85,B 0,C 180,E1 -759.996,E2 -759.996} C_VEL
LIN {X 0,Y 601.407,Z 187.192,A -85,B 0,C 180,E1 -762.671,E2 -762.671} C_VEL
LIN {X 0,Y 601.42,Z 187.191,A -85,B 0,C 180,E1 -765.483,E2 -765.483} C_VEL
LIN {X 0,Y 601.424,Z 187.192,A -85,B 0,C 180,E1 -768.407,E2 -768.407} C_VEL
LIN {X 0,Y 601.427,Z 187.188,A -85,B 0,C 180,E1 -770.876,E2 -770.876} C_VEL
LIN {X 0,Y 601.437,Z 187.194,A -85,B 0,C 180,E1 -773.735,E2 -773.735} C_VEL
LIN {X 0,Y 601.427,Z 187.188,A -85,B 0,C 180,E1 -776.687,E2 -776.687} C_VEL
LIN {X 0,Y 601.408,Z 187.191,A -85,B 0,C 180,E1 -779.058,E2 -779.058} C_VEL
LIN {X 0,Y 601.42,Z 187.193,A -85,B 0,C 180,E1 -781.373,E2 -781.373} C_VEL
LIN {X 0,Y 601.415,Z 187.197,A -85,B 0,C 180,E1 -784.132,E2 -784.132} C_VEL
LIN {X 0,Y 601.444,Z 187.233,A -85,B 0,C 180,E1 -784.523,E2 -784.523} C_VEL
LIN {X 0,Y 601.859,Z 190.744,A -85,B 0,C 180,E1 -784.958,E2 -784.958} C_VEL
LIN {X 0,Y 601.767,Z 214.195,A -85,B 0,C 180,E1 -787.699,E2 -787.699} C_VEL
LIN {X 0,Y 601.668,Z 239.123,A -85,B 0,C 180,E1 -790.555,E2 -790.555} C_VEL
LIN {X 0,Y 601.629,Z 245.872,A -85,B 0,C 180,E1 -791.32,E2 -791.32} C_VEL
LIN {X 0,Y 602.027,Z 250.052,A -85,B 0,C 180,E1 -791.389,E2 -791.389} C_VEL
LIN {X 0,Y 601.887,Z 411.27,A -85,B 0,C 180,E1 -793.377,E2 -793.377} C_VEL
LIN {X 0,Y 601.846,Z 426.903,A -85,B 0,C 180,E1 -793.704,E2 -793.704} C_VEL
LIN {X 0,Y 601.797,Z 441.804,A -85,B 0,C 180,E1 -794.159,E2 -794.159} C_VEL
LIN {X 0,Y 601.719,Z 456.769,A -85,B 0,C 180,E1 -794.764,E2 -794.764} C_VEL
LIN {X 0,Y 601.664,Z 470.24,A -85,B 0,C 180,E1 -795.455,E2 -795.455} C_VEL
LIN {X 0,Y 601.617,Z 483.453,A -85,B 0,C 180,E1 -796.283,E2 -796.283} C_VEL
LIN {X 0,Y 601.531,Z 495.289,A -85,B 0,C 180,E1 -797.175,E2 -797.175} C_VEL
LIN {X 0,Y 601.488,Z 506.751,A -85,B 0,C 180,E1 -798.201,E2 -798.201} C_VEL
LIN {X 0,Y 601.431,Z 516.391,A -85,B 0,C 180,E1 -799.224,E2 -799.224} C_VEL
LIN {X 0,Y 601.428,Z 525.856,A -85,B 0,C 180,E1 -800.415,E2 -800.415} C_VEL
LIN {X 0,Y 601.369,Z 533.731,A -85,B 0,C 180,E1 -801.6,E2 -801.6} C_VEL
LIN {X 0,Y 601.368,Z 541.089,A -85,B 0,C 180,E1 -802.952,E2 -802.952} C_VEL
LIN {X 0,Y 601.373,Z 546.924,A -85,B 0,C 180,E1 -804.299,E2 -804.299} C_VEL
LIN {X 0,Y 601.33,Z 550.384,A -85,B 0,C 180,E1 -805.307,E2 -805.307} C_VEL
LIN {X 0,Y 601.337,Z 553.887,A -85,B 0,C 180,E1 -806.65,E2 -806.65} C_VEL
LIN {X 0,Y 601.343,Z 556.192,A -85,B 0,C 180,E1 -807.991,E2 -807.991} C_VEL
LIN {X 0,Y 601.337,Z 557.35,A -85,B 0,C 180,E1 -809.33,E2 -809.33} C_VEL
LIN {X 0,Y 601.337,Z 557.35,A -85,B 0,C 180,E1 -810.67,E2 -810.67} C_VEL
LIN {X 0,Y 601.343,Z 556.192,A -85,B 0,C 180,E1 -812.009,E2 -812.009} C_VEL
LIN {X 0,Y 601.337,Z 553.886,A -85,B 0,C 180,E1 -813.35,E2 -813.35} C_VEL
LIN {X 0,Y 601.33,Z 550.384,A -85,B 0,C 180,E1 -814.693,E2 -814.693} C_VEL
LIN {X 0,Y 601.357,Z 545.608,A -85,B 0,C 180,E1 -816.038,E2 -816.038} C_VEL
LIN {X 0,Y 601.366,Z 539.426,A -85,B 0,C 180,E1 -817.386,E2 -817.386} C_VEL
LIN {X 0,Y 601.388,Z 531.654,A -85,B 0,C 180,E1 -818.738,E2 -818.738} C_VEL
LIN {X 0,Y 601.427,Z 523.372,A -85,B 0,C 180,E1 -819.925,E2 -819.925} C_VEL
LIN {X 0,Y 601.46,Z 512.93,A -85,B 0,C 180,E1 -821.165,E2 -821.165} C_VEL
LIN {X 0,Y 601.513,Z 503.195,A -85,B 0,C 180,E1 -822.14,E2 -822.14} C_VEL
LIN {X 0,Y 601.57,Z 491.02,A -85,B 0,C 180,E1 -823.168,E2 -823.168} C_VEL
LIN {X 0,Y 601.605,Z 479.081,A -85,B 0,C 180,E1 -824.011,E2 -824.011} C_VEL
LIN {X 0,Y 601.675,Z 465.532,A -85,B 0,C 180,E1 -824.804,E2 -824.804} C_VEL
LIN {X 0,Y 601.772,Z 450.85,A -85,B 0,C 180,E1 -825.495,E2 -825.495} C_VEL
LIN {X 0,Y 601.806,Z 436.628,A -85,B 0,C 180,E1 -826.015,E2 -826.015} C_VEL
LIN {X 0,Y 601.856,Z 421.706,A -85,B 0,C 180,E1 -826.42,E2 -826.42} C_VEL
LIN {X 0,Y 601.867,Z 406.738,A -85,B 0,C 180,E1 -826.689,E2 -826.689} C_VEL
LIN {X 0,Y 601.904,Z 247.485,A -85,B 0,C 180,E1 -828.647,E2 -828.647} C_VEL
LIN {X 0,Y 601.627,Z 245.748,A -85,B 0,C 180,E1 -828.695,E2 -828.695} C_VEL
LIN {X 0,Y 601.751,Z 220.396,A -85,B 0,C 180,E1 -831.585,E2 -831.585} C_VEL
LIN {X 0,Y 601.875,Z 196.311,A -85,B 0,C 180,E1 -834.385,E2 -834.385} C_VEL
LIN {X 0,Y 601.843,Z 189.184,A -85,B 0,C 180,E1 -835.228,E2 -835.228} C_VEL
LIN {X 0,Y 601.434,Z 187.192,A -85,B 0,C 180,E1 -835.501,E2 -835.501} C_VEL
LIN {X 0,Y 601.4,Z 187.197,A -85,B 0,C 180,E1 -837.868,E2 -837.868} C_VEL
LIN {X 0,Y 601.426,Z 187.198,A -85,B 0,C 180,E1 -840.163,E2 -840.163} C_VEL
LIN {X 0,Y 601.413,Z 187.191,A -85,B 0,C 180,E1 -842.714,E2 -842.714} C_VEL
LIN {X 0,Y 601.386,Z 187.192,A -85,B 0,C 180,E1 -845.111,E2 -845.111} C_VEL
LIN {X 0,Y 601.43,Z 187.188,A -85,B 0,C 180,E1 -847.418,E2 -847.418} C_VEL
LIN {X 0,Y 601.406,Z 187.2,A -85,B 0,C 180,E1 -849.994,E2 -849.994} C_VEL
LIN {X 0,Y 601.403,Z 187.192,A -85,B 0,C 180,E1 -852.67,E2 -852.67} C_VEL
LIN {X 0,Y 601.42,Z 187.191,A -85,B 0,C 180,E1 -855.481,E2 -855.481} C_VEL
LIN {X 0,Y 601.416,Z 187.192,A -85,B 0,C 180,E1 -858.406,E2 -858.406} C_VEL
LIN {X 0,Y 601.429,Z 187.187,A -85,B 0,C 180,E1 -860.875,E2 -860.875} C_VEL
LIN {X 0,Y 601.437,Z 187.194,A -85,B 0,C 180,E1 -863.733,E2 -863.733} C_VEL
LIN {X 0,Y 601.425,Z 187.194,A -85,B 0,C 180,E1 -866.064,E2 -866.064} C_VEL
LIN {X 0,Y 601.433,Z 187.187,A -85,B 0,C 180,E1 -868.541,E2 -868.541} C_VEL
LIN {X 0,Y 601.431,Z 187.191,A -85,B 0,C 180,E1 -871.373,E2 -871.373} C_VEL
LIN {X 0,Y 601.4,Z 187.2,A -85,B 0,C 180,E1 -873.636,E2 -873.636} C_VEL
LIN {X 0,Y 601.411,Z 187.189,A -85,B 0,C 180,E1 -876.589,E2 -876.589} C_VEL
LIN {X 0,Y 601.428,Z 187.194,A -85,B 0,C 180,E1 -879.478,E2 -879.478} C_VEL
LIN {X 0,Y 601.392,Z 187.193,A -85,B 0,C 180,E1 -882.312,E2 -882.312} C_VEL
LIN {X 0,Y 601.41,Z 187.19,A -85,B 0,C 180,E1 -884.409,E2 -884.409} C_VEL
LIN {X 0,Y 601.421,Z 187.192,A -85,B 0,C 180,E1 -887.172,E2 -887.172} C_VEL
LIN {X 0,Y 601.425,Z 187.192,A -85,B 0,C 180,E1 -889.905,E2 -889.905} C_VEL
LIN {X 0,Y 601.446,Z 187.185,A -85,B 0,C 180,E1 -892.615,E2 -892.615} C_VEL
LIN {X 0,Y 601.432,Z 187.195,A -85,B 0,C 180,E1 -895.308,E2 -895.308} C_VEL
LIN {X 0,Y 601.414,Z 187.191,A -85,B 0,C 180,E1 -897.991,E2 -897.991} C_VEL
LIN {X 0,Y 601.448,Z 187.186,A -85,B 0,C 180,E1 -900.67,E2 -900.67} C_VEL
LIN {X 0,Y 601.429,Z 187.198,A -85,B 0,C 180,E1 -903.35,E2 -903.35} C_VEL
LIN {X 0,Y 601.4,Z 187.192,A -85,B 0,C 180,E1 -906.037,E2 -906.037} C_VEL
LIN {X 0,Y 601.436,Z 187.189,A -85,B 0,C 180,E1 -908.738,E2 -908.738} C_VEL
LIN {X 0,Y 601.431,Z 187.193,A -85,B 0,C 180,E1 -911.458,E2 -911.458} C_VEL
LIN {X 0,Y 601.404,Z 187.19,A -85,B 0,C 180,E1 -912.386,E2 -912.386} C_VEL
LIN {X 0,Y 600.745,Z 187.28,A -85,B 0,C 180,E1 -912.945,E2 -912.945} C_VEL
LIN {X 0,Y 597.895,Z 187.637,A -85,B 0,C 180,E1 -913.853,E2 -913.853} C_VEL
LIN {X 0,Y 595.482,Z 187.938,A -85,B 0,C 180,E1 -914.583,E2 -914.583} C_VEL
LIN {X 0,Y 594.444,Z 188.068,A -85,B 0,C 180,E1 -915.147,E2 -915.147} C_VEL
LIN {X 0,Y 594.358,Z 188.073,A -85,B 0,C 180,E1 -915.337,E2 -915.337} C_VEL
LIN {X 0,Y 594.373,Z 188.067,A -85,B 0,C 180,E1 -917.904,E2 -917.904} C_VEL
LIN {X 0,Y 594.371,Z 188.074,A -85,B 0,C 180,E1 -920.918,E2 -920.918} C_VEL
LIN {X 0,Y 594.387,Z 188.066,A -85,B 0,C 180,E1 -923.704,E2 -923.704} C_VEL
LIN {X 0,Y 594.383,Z 188.068,A -85,B 0,C 180,E1 -926.7,E2 -926.7} C_VEL
LIN {X 0,Y 594.375,Z 188.077,A -85,B 0,C 180,E1 -928.999,E2 -928.999} C_VEL
LIN {X 0,Y 594.385,Z 188.066,A -85,B 0,C 180,E1 -931.646,E2 -931.646} C_VEL
LIN {X 0,Y 594.392,Z 188.068,A -85,B 0,C 180,E1 -934.579,E2 -934.579} C_VEL
LIN {X 0,Y 594.381,Z 188.072,A -85,B 0,C 180,E1 -937.087,E2 -937.087} C_VEL
LIN {X 0,Y 594.372,Z 188.066,A -85,B 0,C 180,E1 -939.775,E2 -939.775} C_VEL
LIN {X 0,Y 594.363,Z 188.071,A -85,B 0,C 180,E1 -942.376,E2 -942.376} C_VEL
LIN {X 0,Y 594.359,Z 188.072,A -85,B 0,C 180,E1 -945.192,E2 -945.192} C_VEL
LIN {X 0,Y 594.37,Z 188.067,A -85,B 0,C 180,E1 -947.626,E2 -947.626} C_VEL
LIN {X 0,Y 594.369,Z 188.071,A -85,B 0,C 180,E1 -950.32,E2 -950.32} C_VEL
LIN {X 0,Y 594.38,Z 188.072,A -85,B 0,C 180,E1 -952.914,E2 -952.914} C_VEL
LIN {X 0,Y 594.379,Z 188.066,A -85,B 0,C 180,E1 -955.862,E2 -955.862} C_VEL
LIN {X 0,Y 594.378,Z 188.076,A -85,B 0,C 180,E1 -958.651,E2 -958.651} C_VEL
LIN {X 0,Y 594.383,Z 188.069,A -85,B 0,C 180,E1 -961.043,E2 -961.043} C_VEL
LIN {X 0,Y 594.385,Z 188.068,A -85,B 0,C 180,E1 -963.978,E2 -963.978} C_VEL
LIN {X 0,Y 594.385,Z 188.074,A -85,B 0,C 180,E1 -966.296,E2 -966.296} C_VEL
LIN {X 0,Y 594.372,Z 188.121,A -85,B 0,C 180,E1 -967.276,E2 -967.276} C_VEL
LIN {X 0,Y 594.781,Z 191.74,A -85,B 0,C 180,E1 -967.784,E2 -967.784} C_VEL
LIN {X 0,Y 594.669,Z 211.98,A -85,B 0,C 180,E1 -970.497,E2 -970.497} C_VEL
LIN {X 0,Y 594.618,Z 216.924,A -85,B 0,C 180,E1 -971.152,E2 -971.152} C_VEL
LIN {X 0,Y 595.27,Z 221.106,A -85,B 0,C 180,E1 -971.228,E2 -971.228} C_VEL
LIN {X 0,Y 595.094,Z 381.941,A -85,B 0,C 180,E1 -973.237,E2 -973.237} C_VEL
LIN {X 0,Y 595.021,Z 397.696,A -85,B 0,C 180,E1 -973.577,E2 -973.577} C_VEL
LIN {X 0,Y 594.911,Z 413.032,A -85,B 0,C 180,E1 -974.058,E2 -974.058} C_VEL
LIN {X 0,Y 594.857,Z 427.702,A -85,B 0,C 180,E1 -974.672,E2 -974.672} C_VEL
LIN {X 0,Y 594.746,Z 441.003,A -85,B 0,C 180,E1 -975.37,E2 -975.37} C_VEL
LIN {X 0,Y 594.67,Z 453.995,A -85,B 0,C 180,E1 -976.202,E2 -976.202} C_VEL
LIN {X 0,Y 594.552,Z 466.861,A -85,B 0,C 180,E1 -977.195,E2 -977.195} C_VEL
LIN {X 0,Y 594.468,Z 478.065,A -85,B 0,C 180,E1 -978.233,E2 -978.233} C_VEL
LIN {X 0,Y 594.412,Z 488.948,A -85,B 0,C 180,E1 -979.44,E2 -979.44} C_VEL
LIN {X 0,Y 594.356,Z 497.992,A -85,B 0,C 180,E1 -980.643,E2 -980.643} C_VEL
LIN {X 0,Y 594.324,Z 505.486,A -85,B 0,C 180,E1 -981.842,E2 -981.842} C_VEL
LIN {X 0,Y 594.277,Z 512.491,A -85,B 0,C 180,E1 -983.208,E2 -983.208} C_VEL
LIN {X 0,Y 594.273,Z 517.999,A -85,B 0,C 180,E1 -984.571,E2 -984.571} C_VEL
LIN {X 0,Y 594.253,Z 522.171,A -85,B 0,C 180,E1 -985.931,E2 -985.931} C_VEL
LIN {X 0,Y 594.221,Z 525.112,A -85,B 0,C 180,E1 -987.288,E2 -987.288} C_VEL
LIN {X 0,Y 594.244,Z 526.88,A -85,B 0,C 180,E1 -988.645,E2 -988.645} C_VEL
LIN {X 0,Y 594.234,Z 527.496,A -85,B 0,C 180,E1 -990,E2 -990} C_VEL
LIN {X 0,Y 594.246,Z 526.944,A -85,B 0,C 180,E1 -991.355,E2 -991.355} C_VEL
LIN {X 0,Y 594.224,Z 525.26,A -85,B 0,C 180,E1 -992.712,E2 -992.712} C_VEL
LIN {X 0,Y 594.253,Z 522.407,A -85,B 0,C 180,E1 -994.069,E2 -994.069} C_VEL
LIN {X 0,Y 594.273,Z 518.325,A -85,B 0,C 180,E1 -995.429,E2 -995.429} C_VEL
LIN {X 0,Y 594.277,Z 512.916,A -85,B 0,C 180,E1 -996.792,E2 -996.792} C_VEL
LIN {X 0,Y 594.323,Z 506.017,A -85,B 0,C 180,E1 -998.158,E2 -998.158} C_VEL
LIN {X 0,Y 594.339,Z 497.415,A -85,B 0,C 180,E1 -999.529,E2 -999.529} C_VEL
LIN {X 0,Y 594.401,Z 488.266,A -85,B 0,C 180,E1 -1000.732,E2 -1000.732} C_VEL
LIN {X 0,Y 594.466,Z 477.213,A -85,B 0,C 180,E1 -1001.94,E2 -1001.94} C_VEL
LIN {X 0,Y 594.56,Z 465.839,A -85,B 0,C 180,E1 -1002.978,E2 -1002.978} C_VEL
LIN {X 0,Y 594.66,Z 453.457,A -85,B 0,C 180,E1 -1003.925,E2 -1003.925} C_VEL
LIN {X 0,Y 594.728,Z 441.049,A -85,B 0,C 180,E1 -1004.718,E2 -1004.718} C_VEL
LIN {X 0,Y 594.852,Z 427.752,A -85,B 0,C 180,E1 -1005.416,E2 -1005.416} C_VEL
LIN {X 0,Y 594.905,Z 413.082,A -85,B 0,C 180,E1 -1006.03,E2 -1006.03} C_VEL
LIN {X 0,Y 595.033,Z 397.928,A -85,B 0,C 180,E1 -1006.506,E2 -1006.506} C_VEL
LIN {X 0,Y 595.084,Z 382.803,A -85,B 0,C 180,E1 -1006.838,E2 -1006.838} C_VEL
LIN {X 0,Y 595.196,Z 305.688,A -85,B 0,C 180,E1 -1007.812,E2 -1007.812} C_VEL
LIN {X 0,Y 595.152,Z 219.648,A -85,B 0,C 180,E1 -1008.884,E2 -1008.884} C_VEL
LIN {X 0,Y 594.638,Z 216.892,A -85,B 0,C 180,E1 -1008.942,E2 -1008.942} C_VEL
LIN {X 0,Y 594.765,Z 196.455,A -85,B 0,C 180,E1 -1011.67,E2 -1011.67} C_VEL
LIN {X 0,Y 594.755,Z 190.262,A -85,B 0,C 180,E1 -1012.508,E2 -1012.508} C_VEL
LIN {X 0,Y 594.375,Z 188.072,A -85,B 0,C 180,E1 -1012.852,E2 -1012.852} C_VEL
LIN {X 0,Y 594.376,Z 188.072,A -85,B 0,C 180,E1 -1015.192,E2 -1015.192} C_VEL
LIN {X 0,Y 594.385,Z 188.075,A -85,B 0,C 180,E1 -1017.526,E2 -1017.526} C_VEL
LIN {X 0,Y 594.384,Z 188.066,A -85,B 0,C 180,E1 -1020.327,E2 -1020.327} C_VEL
LIN {X 0,Y 594.378,Z 188.069,A -85,B 0,C 180,E1 -1022.949,E2 -1022.949} C_VEL
LIN {X 0,Y 594.354,Z 188.079,A -85,B 0,C 180,E1 -1025.408,E2 -1025.408} C_VEL
LIN {X 0,Y 594.383,Z 188.068,A -85,B 0,C 180,E1 -1027.94,E2 -1027.94} C_VEL
LIN {X 0,Y 594.375,Z 188.068,A -85,B 0,C 180,E1 -1030.822,E2 -1030.822} C_VEL
LIN {X 0,Y 594.378,Z 188.068,A -85,B 0,C 180,E1 -1033.84,E2 -1033.84} C_VEL
LIN {X 0,Y 594.361,Z 188.07,A -85,B 0,C 180,E1 -1036.7,E2 -1036.7} C_VEL
LIN {X 0,Y 594.367,Z 188.074,A -85,B 0,C 180,E1 -1039.433,E2 -1039.433} C_VEL
LIN {X 0,Y 594.384,Z 188.064,A -85,B 0,C 180,E1 -1042.391,E2 -1042.391} C_VEL
LIN {X 0,Y 594.381,Z 188.068,A -85,B 0,C 180,E1 -1044.671,E2 -1044.671} C_VEL
LIN {X 0,Y 594.371,Z 188.077,A -85,B 0,C 180,E1 -1047.088,E2 -1047.088} C_VEL
LIN {X 0,Y 594.394,Z 188.065,A -85,B 0,C 180,E1 -1049.668,E2 -1049.668} C_VEL
LIN {X 0,Y 594.365,Z 188.07,A -85,B 0,C 180,E1 -1052.539,E2 -1052.539} C_VEL
LIN {X 0,Y 594.37,Z 188.073,A -85,B 0,C 180,E1 -1054.807,E2 -1054.807} C_VEL
LIN {X 0,Y 594.357,Z 188.074,A -85,B 0,C 180,E1 -1057.264,E2 -1057.264} C_VEL
LIN {X 0,Y 594.371,Z 188.067,A -85,B 0,C 180,E1 -1059.946,E2 -1059.946} C_VEL
LIN {X 0,Y 594.383,Z 188.074,A -85,B 0,C 180,E1 -1062.806,E2 -1062.806} C_VEL
LIN {X 0,Y 594.379,Z 188.065,A -85,B 0,C 180,E1 -1065.825,E2 -1065.825} C_VEL
LIN {X 0,Y 594.388,Z 188.068,A -85,B 0,C 180,E1 -1068.404,E2 -1068.404} C_VEL
LIN {X 0,Y 594.396,Z 188.068,A -85,B 0,C 180,E1 -1071.158,E2 -1071.158} C_VEL
LIN {X 0,Y 594.357,Z 188.068,A -85,B 0,C 180,E1 -1073.891,E2 -1073.891} C_VEL
LIN {X 0,Y 594.379,Z 188.074,A -85,B 0,C 180,E1 -1076.611,E2 -1076.611} C_VEL
LIN {X 0,Y 594.419,Z 188.061,A -85,B 0,C 180,E1 -1079.322,E2 -1079.322} C_VEL
LIN {X 0,Y 594.383,Z 188.067,A -85,B 0,C 180,E1 -1082.033,E2 -1082.033} C_VEL
LIN {X 0,Y 594.4,Z 188.071,A -85,B 0,C 180,E1 -1084.747,E2 -1084.747} C_VEL
LIN {X 0,Y 594.393,Z 188.064,A -85,B 0,C 180,E1 -1087.473,E2 -1087.473} C_VEL
LIN {X 0,Y 594.385,Z 188.07,A -85,B 0,C 180,E1 -1090.216,E2 -1090.216} C_VEL
LIN {X 0,Y 594.369,Z 188.069,A -85,B 0,C 180,E1 -1092.983,E2 -1092.983} C_VEL
LIN {X 0,Y 594.362,Z 188.069,A -85,B 0,C 180,E1 -1095.781,E2 -1095.781} C_VEL
LIN {X 0,Y 594.38,Z 188.072,A -85,B 0,C 180,E1 -1098.618,E2 -1098.618} C_VEL
LIN {X 0,Y 594.358,Z 188.068,A -85,B 0,C 180,E1 -1101.504,E2 -1101.504} C_VEL
LIN {X 0,Y 594.379,Z 188.074,A -85,B 0,C 180,E1 -1104.446,E2 -1104.446} C_VEL
LIN {X 0,Y 594.382,Z 188.066,A -85,B 0,C 180,E1 -1107.46,E2 -1107.46} C_VEL
LIN {X 0,Y 594.392,Z 188.073,A -85,B 0,C 180,E1 -1110.331,E2 -1110.331} C_VEL
LIN {X 0,Y 594.37,Z 188.067,A -85,B 0,C 180,E1 -1112.951,E2 -1112.951} C_VEL
LIN {X 0,Y 594.375,Z 188.067,A -85,B 0,C 180,E1 -1115.407,E2 -1115.407} C_VEL
LIN {X 0,Y 594.384,Z 188.072,A -85,B 0,C 180,E1 -1117.941,E2 -1117.941} C_VEL
LIN {X 0,Y 594.38,Z 188.065,A -85,B 0,C 180,E1 -1120.824,E2 -1120.824} C_VEL
LIN {X 0,Y 594.36,Z 188.069,A -85,B 0,C 180,E1 -1123.3,E2 -1123.3} C_VEL
LIN {X 0,Y 594.378,Z 188.074,A -85,B 0,C 180,E1 -1126.159,E2 -1126.159} C_VEL
LIN {X 0,Y 594.374,Z 188.067,A -85,B 0,C 180,E1 -1129.178,E2 -1129.178} C_VEL
LIN {X 0,Y 594.383,Z 188.073,A -85,B 0,C 180,E1 -1132.06,E2 -1132.06} C_VEL
LIN {X 0,Y 594.349,Z 188.07,A -85,B 0,C 180,E1 -1134.677,E2 -1134.677} C_VEL
LIN {X 0,Y 594.374,Z 188.067,A -85,B 0,C 180,E1 -1137.089,E2 -1137.089} C_VEL
LIN {X 0,Y 594.383,Z 188.073,A -85,B 0,C 180,E1 -1139.672,E2 -1139.672} C_VEL
LIN {X 0,Y 594.372,Z 188.069,A -85,B 0,C 180,E1 -1142.54,E2 -1142.54} C_VEL
LIN {X 0,Y 594.402,Z 188.208,A -85,B 0,C 180,E1 -1144.316,E2 -1144.316} C_VEL
LIN {X 0,Y 595.046,Z 192.305,A -85,B 0,C 180,E1 -1144.838,E2 -1144.838} C_VEL
LIN {X 0,Y 594.908,Z 215.946,A -85,B 0,C 180,E1 -1147.633,E2 -1147.633} C_VEL
LIN {X 0,Y 594.762,Z 240.684,A -85,B 0,C 180,E1 -1150.5,E2 -1150.5} C_VEL
LIN {X 0,Y 594.7,Z 245.889,A -85,B 0,C 180,E1 -1151.096,E2 -1151.096} C_VEL
LIN {X 0,Y 595.313,Z 249.438,A -85,B 0,C 180,E1 -1151.163,E2 -1151.163} C_VEL
LIN {X 0,Y 595.08,Z 412.397,A -85,B 0,C 180,E1 -1153.199,E2 -1153.199} C_VEL
LIN {X 0,Y 595.019,Z 427.724,A -85,B 0,C 180,E1 -1153.533,E2 -1153.533} C_VEL
LIN {X 0,Y 594.951,Z 443.056,A -85,B 0,C 180,E1 -1154.015,E2 -1154.015} C_VEL
LIN {X 0,Y 594.857,Z 456.772,A -85,B 0,C 180,E1 -1154.584,E2 -1154.584} C_VEL
LIN {X 0,Y 594.741,Z 470.243,A -85,B 0,C 180,E1 -1155.282,E2 -1155.282} C_VEL
LIN {X 0,Y 594.68,Z 482.798,A -85,B 0,C 180,E1 -1156.075,E2 -1156.075} C_VEL
LIN {X 0,Y 594.559,Z 495.29,A -85,B 0,C 180,E1 -1157.022,E2 -1157.022} C_VEL
LIN {X 0,Y 594.465,Z 506.751,A -85,B 0,C 180,E1 -1158.06,E2 -1158.06} C_VEL
LIN {X 0,Y 594.389,Z 516.392,A -85,B 0,C 180,E1 -1159.095,E2 -1159.095} C_VEL
LIN {X 0,Y 594.367,Z 525.857,A -85,B 0,C 180,E1 -1160.3,E2 -1160.3} C_VEL
LIN {X 0,Y 594.312,Z 533.732,A -85,B 0,C 180,E1 -1161.5,E2 -1161.5} C_VEL
LIN {X 0,Y 594.292,Z 541.089,A -85,B 0,C 180,E1 -1162.867,E2 -1162.867} C_VEL
LIN {X 0,Y 594.299,Z 546.925,A -85,B 0,C 180,E1 -1164.231,E2 -1164.231} C_VEL
LIN {X 0,Y 594.232,Z 550.384,A -85,B 0,C 180,E1 -1165.251,E2 -1165.251} C_VEL
LIN {X 0,Y 594.256,Z 553.887,A -85,B 0,C 180,E1 -1166.61,E2 -1166.61} C_VEL
LIN {X 0,Y 594.241,Z 556.193,A -85,B 0,C 180,E1 -1167.967,E2 -1167.967} C_VEL
LIN {X 0,Y 594.237,Z 557.35,A -85,B 0,C 180,E1 -1169.322,E2 -1169.322} C_VEL
LIN {X 0,Y 594.237,Z 557.35,A -85,B 0,C 180,E1 -1170.678,E2 -1170.678} C_VEL
LIN {X 0,Y 594.241,Z 556.192,A -85,B 0,C 180,E1 -1172.033,E2 -1172.033} C_VEL
LIN {X 0,Y 594.256,Z 553.886,A -85,B 0,C 180,E1 -1173.39,E2 -1173.39} C_VEL
LIN {X 0,Y 594.232,Z 550.384,A -85,B 0,C 180,E1 -1174.749,E2 -1174.749} C_VEL
LIN {X 0,Y 594.279,Z 545.609,A -85,B 0,C 180,E1 -1176.11,E2 -1176.11} C_VEL
LIN {X 0,Y 594.287,Z 539.425,A -85,B 0,C 180,E1 -1177.474,E2 -1177.474} C_VEL
LIN {X 0,Y 594.331,Z 531.653,A -85,B 0,C 180,E1 -1178.843,E2 -1178.843} C_VEL
LIN {X 0,Y 594.387,Z 523.371,A -85,B 0,C 180,E1 -1180.044,E2 -1180.044} C_VEL
LIN {X 0,Y 594.434,Z 513.557,A -85,B 0,C 180,E1 -1181.231,E2 -1181.231} C_VEL
LIN {X 0,Y 594.53,Z 503.194,A -85,B 0,C 180,E1 -1182.285,E2 -1182.285} C_VEL
LIN {X 0,Y 594.581,Z 491.021,A -85,B 0,C 180,E1 -1183.326,E2 -1183.326} C_VEL
LIN {X 0,Y 594.693,Z 479.078,A -85,B 0,C 180,E1 -1184.177,E2 -1184.177} C_VEL
LIN {X 0,Y 594.776,Z 465.529,A -85,B 0,C 180,E1 -1184.98,E2 -1184.98} C_VEL
LIN {X 0,Y 594.913,Z 450.847,A -85,B 0,C 180,E1 -1185.678,E2 -1185.678} C_VEL
LIN {X 0,Y 594.979,Z 436.628,A -85,B 0,C 180,E1 -1186.204,E2 -1186.204} C_VEL
LIN {X 0,Y 595.045,Z 422.134,A -85,B 0,C 180,E1 -1186.603,E2 -1186.603} C_VEL
LIN {X 0,Y 595.067,Z 406.738,A -85,B 0,C 180,E1 -1186.886,E2 -1186.886} C_VEL
LIN {X 0,Y 595.217,Z 248.554,A -85,B 0,C 180,E1 -1188.851,E2 -1188.851} C_VEL
LIN {X 0,Y 594.731,Z 245.804,A -85,B 0,C 180,E1 -1188.913,E2 -1188.913} C_VEL
LIN {X 0,Y 594.894,Z 220.396,A -85,B 0,C 180,E1 -1191.847,E2 -1191.847} C_VEL
LIN {X 0,Y 595.045,Z 197.239,A -85,B 0,C 180,E1 -1194.573,E2 -1194.573} C_VEL
LIN {X 0,Y 594.983,Z 190.744,A -85,B 0,C 180,E1 -1195.352,E2 -1195.352} C_VEL
LIN {X 0,Y 594.391,Z 188.072,A -85,B 0,C 180,E1 -1195.708,E2 -1195.708} C_VEL
LIN {X 0,Y 594.369,Z 188.077,A -85,B 0,C 180,E1 -1198.227,E2 -1198.227} C_VEL
LIN {X 0,Y 594.377,Z 188.07,A -85,B 0,C 180,E1 -1200.559,E2 -1200.559} C_VEL
LIN {X 0,Y 594.375,Z 188.066,A -85,B 0,C 180,E1 -1202.95,E2 -1202.95} C_VEL
LIN {X 0,Y 594.35,Z 188.07,A -85,B 0,C 180,E1 -1205.408,E2 -1205.408} C_VEL
LIN {X 0,Y 594.384,Z 188.073,A -85,B 0,C 180,E1 -1207.94,E2 -1207.94} C_VEL
LIN {X 0,Y 594.374,Z 188.067,A -85,B 0,C 180,E1 -1210.822,E2 -1210.822} C_VEL
LIN {X 0,Y 594.378,Z 188.073,A -85,B 0,C 180,E1 -1213.841,E2 -1213.841} C_VEL
LIN {X 0,Y 594.36,Z 188.068,A -85,B 0,C 180,E1 -1216.7,E2 -1216.7} C_VEL
LIN {X 0,Y 594.382,Z 188.068,A -85,B 0,C 180,E1 -1219.434,E2 -1219.434} C_VEL
LIN {X 0,Y 594.384,Z 188.067,A -85,B 0,C 180,E1 -1222.391,E2 -1222.391} C_VEL
LIN {X 0,Y 594.377,Z 188.066,A -85,B 0,C 180,E1 -1224.671,E2 -1224.671} C_VEL
LIN {X 0,Y 594.371,Z 188.067,A -85,B 0,C 180,E1 -1227.088,E2 -1227.088} C_VEL
LIN {X 0,Y 594.393,Z 188.072,A -85,B 0,C 180,E1 -1229.669,E2 -1229.669} C_VEL
LIN {X 0,Y 594.382,Z 188.065,A -85,B 0,C 180,E1 -1232.54,E2 -1232.54} C_VEL
LIN {X 0,Y 594.389,Z 188.072,A -85,B 0,C 180,E1 -1235.563,E2 -1235.563} C_VEL
LIN {X 0,Y 594.358,Z 188.067,A -85,B 0,C 180,E1 -1238.496,E2 -1238.496} C_VEL
LIN {X 0,Y 594.38,Z 188.071,A -85,B 0,C 180,E1 -1241.382,E2 -1241.382} C_VEL
LIN {X 0,Y 594.363,Z 188.069,A -85,B 0,C 180,E1 -1244.219,E2 -1244.219} C_VEL
LIN {X 0,Y 594.368,Z 188.069,A -85,B 0,C 180,E1 -1247.017,E2 -1247.017} C_VEL
LIN {X 0,Y 594.386,Z 188.071,A -85,B 0,C 180,E1 -1249.784,E2 -1249.784} C_VEL
LIN {X 0,Y 594.394,Z 188.064,A -85,B 0,C 180,E1 -1252.527,E2 -1252.527} C_VEL
LIN {X 0,Y 594.399,Z 188.07,A -85,B 0,C 180,E1 -1255.253,E2 -1255.253} C_VEL
LIN {X 0,Y 594.384,Z 188.067,A -85,B 0,C 180,E1 -1257.967,E2 -1257.967} C_VEL
LIN {X 0,Y 594.418,Z 188.061,A -85,B 0,C 180,E1 -1260.678,E2 -1260.678} C_VEL
LIN {X 0,Y 594.38,Z 188.075,A -85,B 0,C 180,E1 -1263.389,E2 -1263.389} C_VEL
LIN {X 0,Y 594.357,Z 188.069,A -85,B 0,C 180,E1 -1266.109,E2 -1266.109} C_VEL
LIN {X 0,Y 594.397,Z 188.067,A -85,B 0,C 180,E1 -1268.842,E2 -1268.842} C_VEL
LIN {X 0,Y 594.388,Z 188.069,A -85,B 0,C 180,E1 -1271.596,E2 -1271.596} C_VEL
LIN {X 0,Y 594.381,Z 188.066,A -85,B 0,C 180,E1 -1274.377,E2 -1274.377} C_VEL
LIN {X 0,Y 594.358,Z 188.073,A -85,B 0,C 180,E1 -1275.337,E2 -1275.337} C_VEL
LIN {X 0,Y 593.688,Z 188.154,A -85,B 0,C 180,E1 -1275.903,E2 -1275.903} C_VEL
LIN {X 0,Y 590.833,Z 188.512,A -85,B 0,C 180,E1 -1276.821,E2 -1276.821} C_VEL
LIN {X 0,Y 588.426,Z 188.811,A -85,B 0,C 180,E1 -1277.56,E2 -1277.56} C_VEL
LIN {X 0,Y 587.398,Z 188.936,A -85,B 0,C 180,E1 -1278.13,E2 -1278.13} C_VEL
LIN {X 0,Y 587.317,Z 188.946,A -85,B 0,C 180,E1 -1278.323,E2 -1278.323} C_VEL
LIN {X 0,Y 587.32,Z 188.954,A -85,B 0,C 180,E1 -1281.038,E2 -1281.038} C_VEL
LIN {X 0,Y 587.316,Z 188.952,A -85,B 0,C 180,E1 -1283.259,E2 -1283.259} C_VEL
LIN {X 0,Y 587.329,Z 188.944,A -85,B 0,C 180,E1 -1285.517,E2 -1285.517} C_VEL
LIN {X 0,Y 587.341,Z 188.942,A -85,B 0,C 180,E1 -1287.818,E2 -1287.818} C_VEL
LIN {X 0,Y 587.344,Z 188.945,A -85,B 0,C 180,E1 -1290.513,E2 -1290.513} C_VEL
LIN {X 0,Y 587.328,Z 188.947,A -85,B 0,C 180,E1 -1293.397,E2 -1293.397} C_VEL
LIN {X 0,Y 587.351,Z 188.941,A -85,B 0,C 180,E1 -1295.896,E2 -1295.896} C_VEL
LIN {X 0,Y 587.329,Z 188.948,A -85,B 0,C 180,E1 -1298.48,E2 -1298.48} C_VEL
LIN {X 0,Y 587.332,Z 188.948,A -85,B 0,C 180,E1 -1301.157,E2 -1301.157} C_VEL
LIN {X 0,Y 587.321,Z 188.946,A -85,B 0,C 180,E1 -1304.114,E2 -1304.114} C_VEL
LIN {X 0,Y 587.32,Z 188.951,A -85,B 0,C 180,E1 -1306.995,E2 -1306.995} C_VEL
LIN {X 0,Y 587.31,Z 188.947,A -85,B 0,C 180,E1 -1309.746,E2 -1309.746} C_VEL
LIN {X 0,Y 587.342,Z 188.948,A -85,B 0,C 180,E1 -1312.393,E2 -1312.393} C_VEL
LIN {X 0,Y 587.359,Z 188.941,A -85,B 0,C 180,E1 -1315.781,E2 -1315.781} C_VEL
LIN {X 0,Y 587.346,Z 188.947,A -85,B 0,C 180,E1 -1318.232,E2 -1318.232} C_VEL
LIN {X 0,Y 587.349,Z 188.948,A -85,B 0,C 180,E1 -1320.867,E2 -1320.867} C_VEL
LIN {X 0,Y 587.359,Z 188.942,A -85,B 0,C 180,E1 -1323.819,E2 -1323.819} C_VEL
LIN {X 0,Y 587.334,Z 188.948,A -85,B 0,C 180,E1 -1325.994,E2 -1325.994} C_VEL
LIN {X 0,Y 587.355,Z 189.102,A -85,B 0,C 180,E1 -1327.124,E2 -1327.124} C_VEL
LIN {X 0,Y 587.875,Z 193.093,A -85,B 0,C 180,E1 -1327.694,E2 -1327.694} C_VEL
LIN {X 0,Y 587.738,Z 214.352,A -85,B 0,C 180,E1 -1330.576,E2 -1330.576} C_VEL
LIN {X 0,Y 587.676,Z 216.847,A -85,B 0,C 180,E1 -1330.91,E2 -1330.91} C_VEL
LIN {X 0,Y 588.578,Z 221.959,A -85,B 0,C 180,E1 -1331.016,E2 -1331.016} C_VEL
LIN {X 0,Y 588.294,Z 382.512,A -85,B 0,C 180,E1 -1333.047,E2 -1333.047} C_VEL
LIN {X 0,Y 588.203,Z 398.492,A -85,B 0,C 180,E1 -1333.403,E2 -1333.403} C_VEL
LIN {X 0,Y 588.068,Z 413.046,A -85,B 0,C 180,E1 -1333.868,E2 -1333.868} C_VEL
LIN {X 0,Y 587.995,Z 427.712,A -85,B 0,C 180,E1 -1334.489,E2 -1334.489} C_VEL
LIN {X 0,Y 587.848,Z 441.016,A -85,B 0,C 180,E1 -1335.194,E2 -1335.194} C_VEL
LIN {X 0,Y 587.734,Z 454.18,A -85,B 0,C 180,E1 -1336.048,E2 -1336.048} C_VEL
LIN {X 0,Y 587.558,Z 466.87,A -85,B 0,C 180,E1 -1337.04,E2 -1337.04} C_VEL
LIN {X 0,Y 587.472,Z 478.07,A -85,B 0,C 180,E1 -1338.091,E2 -1338.091} C_VEL
LIN {X 0,Y 587.382,Z 488.953,A -85,B 0,C 180,E1 -1339.312,E2 -1339.312} C_VEL
LIN {X 0,Y 587.285,Z 497.995,A -85,B 0,C 180,E1 -1340.529,E2 -1340.529} C_VEL
LIN {X 0,Y 587.258,Z 505.489,A -85,B 0,C 180,E1 -1341.743,E2 -1341.743} C_VEL
LIN {X 0,Y 587.208,Z 512.493,A -85,B 0,C 180,E1 -1343.126,E2 -1343.126} C_VEL
LIN {X 0,Y 587.198,Z 518.001,A -85,B 0,C 180,E1 -1344.506,E2 -1344.506} C_VEL
LIN {X 0,Y 587.169,Z 522.173,A -85,B 0,C 180,E1 -1345.882,E2 -1345.882} C_VEL
LIN {X 0,Y 587.127,Z 525.114,A -85,B 0,C 180,E1 -1347.256,E2 -1347.256} C_VEL
LIN {X 0,Y 587.143,Z 526.88,A -85,B 0,C 180,E1 -1348.628,E2 -1348.628} C_VEL
LIN {X 0,Y 587.135,Z 527.496,A -85,B 0,C 180,E1 -1350,E2 -1350} C_VEL
LIN {X 0,Y 587.146,Z 526.943,A -85,B 0,C 180,E1 -1351.372,E2 -1351.372} C_VEL
LIN {X 0,Y 587.129,Z 525.26,A -85,B 0,C 180,E1 -1352.744,E2 -1352.744} C_VEL
LIN {X 0,Y 587.169,Z 522.406,A -85,B 0,C 180,E1 -1354.118,E2 -1354.118} C_VEL
LIN {X 0,Y 587.198,Z 518.324,A -85,B 0,C 180,E1 -1355.494,E2 -1355.494} C_VEL
LIN {X 0,Y 587.208,Z 512.913,A -85,B 0,C 180,E1 -1356.874,E2 -1356.874} C_VEL
LIN {X 0,Y 587.254,Z 506.014,A -85,B 0,C 180,E1 -1358.257,E2 -1358.257} C_VEL
LIN {X 0,Y 587.286,Z 497.41,A -85,B 0,C 180,E1 -1359.644,E2 -1359.644} C_VEL
LIN {X 0,Y 587.367,Z 488.261,A -85,B 0,C 180,E1 -1360.862,E2 -1360.862} C_VEL
LIN {X 0,Y 587.446,Z 478.933,A -85,B 0,C 180,E1 -1361.91,E2 -1361.91} C_VEL
LIN {X 0,Y 587.588,Z 466.892,A -85,B 0,C 180,E1 -1363.047,E2 -1363.047} C_VEL
LIN {X 0,Y 587.71,Z 453.8,A -85,B 0,C 180,E1 -1364.069,E2 -1364.069} C_VEL
LIN {X 0,Y 587.822,Z 441.042,A -85,B 0,C 180,E1 -1364.895,E2 -1364.895} C_VEL
LIN {X 0,Y 587.987,Z 427.739,A -85,B 0,C 180,E1 -1365.6,E2 -1365.6} C_VEL
LIN {X 0,Y 588.071,Z 413.065,A -85,B 0,C 180,E1 -1366.221,E2 -1366.221} C_VEL
LIN {X 0,Y 588.218,Z 397.992,A -85,B 0,C 180,E1 -1366.701,E2 -1366.701} C_VEL
LIN {X 0,Y 588.292,Z 382.404,A -85,B 0,C 180,E1 -1367.045,E2 -1367.045} C_VEL
LIN {X 0,Y 588.589,Z 221.631,A -85,B 0,C 180,E1 -1369.077,E2 -1369.077} C_VEL
LIN {X 0,Y 587.696,Z 216.863,A -85,B 0,C 180,E1 -1369.178,E2 -1369.178} C_VEL
LIN {X 0,Y 587.868,Z 196.45,A -85,B 0,C 180,E1 -1371.937,E2 -1371.937} C_VEL
LIN {X 0,Y 587.797,Z 191.38,A -85,B 0,C 180,E1 -1372.635,E2 -1372.635} C_VEL
LIN {X 0,Y 587.333,Z 188.951,A -85,B 0,C 180,E1 -1373.025,E2 -1373.025} C_VEL
LIN {X 0,Y 587.336,Z 188.954,A -85,B 0,C 180,E1 -1375.516,E2 -1375.516} C_VEL
LIN {X 0,Y 587.346,Z 188.948,A -85,B 0,C 180,E1 -1377.817,E2 -1377.817} C_VEL
LIN {X 0,Y 587.334,Z 188.944,A -85,B 0,C 180,E1 -1380.509,E2 -1380.509} C_VEL
LIN {X 0,Y 587.339,Z 188.948,A -85,B 0,C 180,E1 -1383.111,E2 -1383.111} C_VEL
LIN {X 0,Y 587.326,Z 188.953,A -85,B 0,C 180,E1 -1385.541,E2 -1385.541} C_VEL
LIN {X 0,Y 587.337,Z 188.947,A -85,B 0,C 180,E1 -1387.838,E2 -1387.838} C_VEL
LIN {X 0,Y 587.315,Z 188.946,A -85,B 0,C 180,E1 -1390.253,E2 -1390.253} C_VEL
LIN {X 0,Y 587.318,Z 188.95,A -85,B 0,C 180,E1 -1393.005,E2 -1393.005} C_VEL
LIN {X 0,Y 587.321,Z 188.947,A -85,B 0,C 180,E1 -1395.886,E2 -1395.886} C_VEL
LIN {X 0,Y 587.331,Z 188.947,A -85,B 0,C 180,E1 -1398.842,E2 -1398.842} C_VEL
LIN {X 0,Y 587.328,Z 188.948,A -85,B 0,C 180,E1 -1401.52,E2 -1401.52} C_VEL
LIN {X 0,Y 587.347,Z 188.942,A -85,B 0,C 180,E1 -1404.454,E2 -1404.454} C_VEL
LIN {X 0,Y 587.332,Z 188.95,A -85,B 0,C 180,E1 -1406.887,E2 -1406.887} C_VEL
LIN {X 0,Y 587.344,Z 188.945,A -85,B 0,C 180,E1 -1409.487,E2 -1409.487} C_VEL
LIN {X 0,Y 587.343,Z 188.943,A -85,B 0,C 180,E1 -1412.306,E2 -1412.306} C_VEL
LIN {X 0,Y 587.328,Z 188.946,A -85,B 0,C 180,E1 -1414.483,E2 -1414.483} C_VEL
LIN {X 0,Y 587.311,Z 188.954,A -85,B 0,C 180,E1 -1417.13,E2 -1417.13} C_VEL
LIN {X 0,Y 587.325,Z 188.945,A -85,B 0,C 180,E1 -1419.695,E2 -1419.695} C_VEL
LIN {X 0,Y 587.35,Z 188.946,A -85,B 0,C 180,E1 -1422.594,E2 -1422.594} C_VEL
LIN {X 0,Y 587.355,Z 188.94,A -85,B 0,C 180,E1 -1425.739,E2 -1425.739} C_VEL
LIN {X 0,Y 587.352,Z 188.95,A -85,B 0,C 180,E1 -1428.858,E2 -1428.858} C_VEL
LIN {X 0,Y 587.361,Z 188.94,A -85,B 0,C 180,E1 -1431.745,E2 -1431.745} C_VEL
LIN {X 0,Y 587.357,Z 188.947,A -85,B 0,C 180,E1 -1434.507,E2 -1434.507} C_VEL
LIN {X 0,Y 587.374,Z 188.94,A -85,B 0,C 180,E1 -1437.257,E2 -1437.257} C_VEL
LIN {X 0,Y 587.369,Z 188.939,A -85,B 0,C 180,E1 -1440,E2 -1440} C_VEL
LIN {X 0,Y 587.374,Z 188.946,A -85,B 0,C 180,E1 -1442.743,E2 -1442.743} C_VEL
LIN {X 0,Y 587.353,Z 188.941,A -85,B 0,C 180,E1 -1445.493,E2 -1445.493} C_VEL
LIN {X 0,Y 587.361,Z 188.945,A -85,B 0,C 180,E1 -1448.255,E2 -1448.255} C_VEL
LIN {X 0,Y 587.352,Z 188.943,A -85,B 0,C 180,E1 -1451.141,E2 -1451.141} C_VEL
LIN {X 0,Y 587.355,Z 188.947,A -85,B 0,C 180,E1 -1454.261,E2 -1454.261} C_VEL
LIN {X 0,Y 587.351,Z 188.941,A -85,B 0,C 180,E1 -1457.406,E2 -1457.406} C_VEL
LIN {X 0,Y 587.326,Z 188.954,A -85,B 0,C 180,E1 -1460.305,E2 -1460.305} C_VEL
LIN {X 0,Y 587.315,Z 188.946,A -85,B 0,C 180,E1 -1463.259,E2 -1463.259} C_VEL
LIN {X 0,Y 587.324,Z 188.945,A -85,B 0,C 180,E1 -1465.517,E2 -1465.517} C_VEL
LIN {X 0,Y 587.341,Z 188.946,A -85,B 0,C 180,E1 -1467.818,E2 -1467.818} C_VEL
LIN {X 0,Y 587.343,Z 188.948,A -85,B 0,C 180,E1 -1470.513,E2 -1470.513} C_VEL
LIN {X 0,Y 587.325,Z 188.944,A -85,B 0,C 180,E1 -1473.397,E2 -1473.397} C_VEL
LIN {X 0,Y 587.349,Z 188.947,A -85,B 0,C 180,E1 -1475.896,E2 -1475.896} C_VEL
LIN {X 0,Y 587.326,Z 188.948,A -85,B 0,C 180,E1 -1478.48,E2 -1478.48} C_VEL
LIN {X 0,Y 587.332,Z 188.942,A -85,B 0,C 180,E1 -1481.157,E2 -1481.157} C_VEL
LIN {X 0,Y 587.32,Z 188.954,A -85,B 0,C 180,E1 -1484.114,E2 -1484.114} C_VEL
LIN {X 0,Y 587.314,Z 188.946,A -85,B 0,C 180,E1 -1486.995,E2 -1486.995} C_VEL
LIN {X 0,Y 587.313,Z 188.953,A -85,B 0,C 180,E1 -1489.747,E2 -1489.747} C_VEL
LIN {X 0,Y 587.341,Z 188.945,A -85,B 0,C 180,E1 -1492.393,E2 -1492.393} C_VEL
LIN {X 0,Y 587.32,Z 188.945,A -85,B 0,C 180,E1 -1494.945,E2 -1494.945} C_VEL
LIN {X 0,Y 587.333,Z 188.947,A -85,B 0,C 180,E1 -1497.421,E2 -1497.421} C_VEL
LIN {X 0,Y 587.331,Z 188.954,A -85,B 0,C 180,E1 -1499.831,E2 -1499.831} C_VEL
LIN {X 0,Y 587.339,Z 188.948,A -85,B 0,C 180,E1 -1502.31,E2 -1502.31} C_VEL
LIN {X 0,Y 587.357,Z 189.063,A -85,B 0,C 180,E1 -1504.091,E2 -1504.091} C_VEL
LIN {X 0,Y 588.255,Z 194.022,A -85,B 0,C 180,E1 -1504.735,E2 -1504.735} C_VEL
LIN {X 0,Y 588.056,Z 218.835,A -85,B 0,C 180,E1 -1507.701,E2 -1507.701} C_VEL
LIN {X 0,Y 587.84,Z 243.367,A -85,B 0,C 180,E1 -1510.573,E2 -1510.573} C_VEL
LIN {X 0,Y 587.814,Z 246.05,A -85,B 0,C 180,E1 -1510.871,E2 -1510.871} C_VEL
LIN {X 0,Y 588.594,Z 250.58,A -85,B 0,C 180,E1 -1510.954,E2 -1510.954} C_VEL
LIN {X 0,Y 588.3,Z 412.377,A -85,B 0,C 180,E1 -1512.999,E2 -1512.999} C_VEL
LIN {X 0,Y 588.208,Z 427.722,A -85,B 0,C 180,E1 -1513.337,E2 -1513.337} C_VEL
LIN {X 0,Y 588.084,Z 443.054,A -85,B 0,C 180,E1 -1513.824,E2 -1513.824} C_VEL
LIN {X 0,Y 587.996,Z 456.775,A -85,B 0,C 180,E1 -1514.4,E2 -1514.4} C_VEL
LIN {X 0,Y 587.84,Z 470.246,A -85,B 0,C 180,E1 -1515.106,E2 -1515.106} C_VEL
LIN {X 0,Y 587.74,Z 483.119,A -85,B 0,C 180,E1 -1515.93,E2 -1515.93} C_VEL
LIN {X 0,Y 587.582,Z 495.291,A -85,B 0,C 180,E1 -1516.865,E2 -1516.865} C_VEL
LIN {X 0,Y 587.453,Z 506.752,A -85,B 0,C 180,E1 -1517.915,E2 -1517.915} C_VEL
LIN {X 0,Y 587.349,Z 516.392,A -85,B 0,C 180,E1 -1518.963,E2 -1518.963} C_VEL
LIN {X 0,Y 587.305,Z 525.858,A -85,B 0,C 180,E1 -1520.182,E2 -1520.182} C_VEL
LIN {X 0,Y 587.265,Z 533.733,A -85,B 0,C 180,E1 -1521.397,E2 -1521.397} C_VEL
LIN {X 0,Y 587.215,Z 541.089,A -85,B 0,C 180,E1 -1522.781,E2 -1522.781} C_VEL
LIN {X 0,Y 587.227,Z 546.924,A -85,B 0,C 180,E1 -1524.161,E2 -1524.161} C_VEL
LIN {X 0,Y 587.136,Z 550.385,A -85,B 0,C 180,E1 -1525.194,E2 -1525.194} C_VEL
LIN {X 0,Y 587.179,Z 553.888,A -85,B 0,C 180,E1 -1526.569,E2 -1526.569} C_VEL
LIN {X 0,Y 587.14,Z 556.193,A -85,B 0,C 180,E1 -1527.942,E2 -1527.942} C_VEL
LIN {X 0,Y 587.138,Z 557.35,A -85,B 0,C 180,E1 -1529.314,E2 -1529.314} C_VEL
LIN {X 0,Y 587.138,Z 557.349,A -85,B 0,C 180,E1 -1530.686,E2 -1530.686} C_VEL
LIN {X 0,Y 587.14,Z 556.192,A -85,B 0,C 180,E1 -1532.058,E2 -1532.058} C_VEL
LIN {X 0,Y 587.179,Z 553.886,A -85,B 0,C 180,E1 -1533.431,E2 -1533.431} C_VEL
LIN {X 0,Y 587.136,Z 550.385,A -85,B 0,C 180,E1 -1534.806,E2 -1534.806} C_VEL
LIN {X 0,Y 587.18,Z 545.609,A -85,B 0,C 180,E1 -1536.184,E2 -1536.184} C_VEL
LIN {X 0,Y 587.23,Z 539.425,A -85,B 0,C 180,E1 -1537.565,E2 -1537.565} C_VEL
LIN {X 0,Y 587.266,Z 531.652,A -85,B 0,C 180,E1 -1538.95,E2 -1538.95} C_VEL
LIN {X 0,Y 587.351,Z 523.371,A -85,B 0,C 180,E1 -1540.165,E2 -1540.165} C_VEL
LIN {X 0,Y 587.399,Z 513.397,A -85,B 0,C 180,E1 -1541.385,E2 -1541.385} C_VEL
LIN {X 0,Y 587.522,Z 503.193,A -85,B 0,C 180,E1 -1542.434,E2 -1542.434} C_VEL
LIN {X 0,Y 587.629,Z 491.022,A -85,B 0,C 180,E1 -1543.486,E2 -1543.486} C_VEL
LIN {X 0,Y 587.774,Z 478.063,A -85,B 0,C 180,E1 -1544.416,E2 -1544.416} C_VEL
LIN {X 0,Y 587.927,Z 463.874,A -85,B 0,C 180,E1 -1545.247,E2 -1545.247} C_VEL
LIN {X 0,Y 588.059,Z 449.805,A -85,B 0,C 180,E1 -1545.91,E2 -1545.91} C_VEL
LIN {X 0,Y 588.175,Z 435.315,A -85,B 0,C 180,E1 -1546.441,E2 -1546.441} C_VEL
LIN {X 0,Y 588.278,Z 420.291,A -85,B 0,C 180,E1 -1546.844,E2 -1546.844} C_VEL
LIN {X 0,Y 588.321,Z 405.097,A -85,B 0,C 180,E1 -1547.11,E2 -1547.11} C_VEL
LIN {X 0,Y 588.505,Z 249.436,A -85,B 0,C 180,E1 -1549.063,E2 -1549.063} C_VEL
LIN {X 0,Y 587.804,Z 245.775,A -85,B 0,C 180,E1 -1549.148,E2 -1549.148} C_VEL
LIN {X 0,Y 588.031,Z 220.396,A -85,B 0,C 180,E1 -1552.115,E2 -1552.115} C_VEL
LIN {X 0,Y 588.237,Z 197.144,A -85,B 0,C 180,E1 -1554.888,E2 -1554.888} C_VEL
LIN {X 0,Y 588.122,Z 192.305,A -85,B 0,C 180,E1 -1555.479,E2 -1555.479} C_VEL
LIN {X 0,Y 587.344,Z 188.952,A -85,B 0,C 180,E1 -1555.949,E2 -1555.949} C_VEL
LIN {X 0,Y 587.317,Z 188.95,A -85,B 0,C 180,E1 -1558.597,E2 -1558.597} C_VEL
LIN {X 0,Y 587.325,Z 188.945,A -85,B 0,C 180,E1 -1560.966,E2 -1560.966} C_VEL
LIN {X 0,Y 587.334,Z 188.943,A -85,B 0,C 180,E1 -1563.396,E2 -1563.396} C_VEL
LIN {X 0,Y 587.313,Z 188.952,A -85,B 0,C 180,E1 -1565.898,E2 -1565.898} C_VEL
LIN {X 0,Y 587.328,Z 188.948,A -85,B 0,C 180,E1 -1568.478,E2 -1568.478} C_VEL
LIN {X 0,Y 587.333,Z 188.944,A -85,B 0,C 180,E1 -1571.156,E2 -1571.156} C_VEL
LIN {X 0,Y 587.329,Z 188.952,A -85,B 0,C 180,E1 -1574.114,E2 -1574.114} C_VEL
LIN {X 0,Y 587.309,Z 188.946,A -85,B 0,C 180,E1 -1576.993,E2 -1576.993} C_VEL
LIN {X 0,Y 587.322,Z 188.952,A -85,B 0,C 180,E1 -1579.746,E2 -1579.746} C_VEL
LIN {X 0,Y 587.339,Z 188.945,A -85,B 0,C 180,E1 -1582.392,E2 -1582.392} C_VEL
LIN {X 0,Y 587.343,Z 188.942,A -85,B 0,C 180,E1 -1584.946,E2 -1584.946} C_VEL
LIN {X 0,Y 587.333,Z 188.947,A -85,B 0,C 180,E1 -1587.421,E2 -1587.421} C_VEL
LIN {X 0,Y 587.338,Z 188.952,A -85,B 0,C 180,E1 -1589.83,E2 -1589.83} C_VEL
LIN {X 0,Y 587.343,Z 188.944,A -85,B 0,C 180,E1 -1592.306,E2 -1592.306} C_VEL
LIN {X 0,Y 587.342,Z 188.945,A -85,B 0,C 180,E1 -1595.241,E2 -1595.241} C_VEL
LIN {X 0,Y 587.315,Z 188.946,A -85,B 0,C 180,E1 -1598.225,E2 -1598.225} C_VEL
LIN {X 0,Y 587.344,Z 188.945,A -85,B 0,C 180,E1 -1601.151,E2 -1601.151} C_VEL
LIN {X 0,Y 587.347,Z 188.947,A -85,B 0,C 180,E1 -1603.311,E2 -1603.311} C_VEL
LIN {X 0,Y 587.353,Z 188.943,A -85,B 0,C 180,E1 -1606.154,E2 -1606.154} C_VEL
LIN {X 0,Y 587.338,Z 188.945,A -85,B 0,C 180,E1 -1608.962,E2 -1608.962} C_VEL
LIN {X 0,Y 587.362,Z 188.946,A -85,B 0,C 180,E1 -1611.745,E2 -1611.745} C_VEL
LIN {X 0,Y 587.354,Z 188.941,A -85,B 0,C 180,E1 -1614.507,E2 -1614.507} C_VEL
LIN {X 0,Y 587.375,Z 188.945,A -85,B 0,C 180,E1 -1617.257,E2 -1617.257} C_VEL
LIN {X 0,Y 587.37,Z 188.94,A -85,B 0,C 180,E1 -1620,E2 -1620} C_VEL
LIN {X 0,Y 587.373,Z 188.94,A -85,B 0,C 180,E1 -1622.743,E2 -1622.743} C_VEL
LIN {X 0,Y 587.356,Z 188.948,A -85,B 0,C 180,E1 -1625.493,E2 -1625.493} C_VEL
LIN {X 0,Y 587.362,Z 188.939,A -85,B 0,C 180,E1 -1628.255,E2 -1628.255} C_VEL
LIN {X 0,Y 587.352,Z 188.95,A -85,B 0,C 180,E1 -1631.142,E2 -1631.142} C_VEL
LIN {X 0,Y 587.355,Z 188.941,A -85,B 0,C 180,E1 -1634.261,E2 -1634.261} C_VEL
LIN {X 0,Y 587.351,Z 188.947,A -85,B 0,C 180,E1 -1637.406,E2 -1637.406} C_VEL
LIN {X 0,Y 587.317,Z 188.946,A -85,B 0,C 180,E1 -1638.323,E2 -1638.323} C_VEL
LIN {X 0,Y 586.663,Z 189.034,A -85,B 0,C 180,E1 -1638.895,E2 -1638.895} C_VEL
LIN {X 0,Y 583.829,Z 189.392,A -85,B 0,C 180,E1 -1639.824,E2 -1639.824} C_VEL
LIN {X 0,Y 581.418,Z 189.693,A -85,B 0,C 180,E1 -1640.571,E2 -1640.571} C_VEL
LIN {X 0,Y 580.367,Z 189.821,A -85,B 0,C 180,E1 -1641.147,E2 -1641.147} C_VEL
LIN {X 0,Y 580.273,Z 189.829,A -85,B 0,C 180,E1 -1641.342,E2 -1641.342} C_VEL
LIN {X 0,Y 580.294,Z 189.821,A -85,B 0,C 180,E1 -1644.317,E2 -1644.317} C_VEL
LIN {X 0,Y 580.274,Z 189.823,A -85,B 0,C 180,E1 -1646.624,E2 -1646.624} C_VEL
LIN {X 0,Y 580.298,Z 189.825,A -85,B 0,C 180,E1 -1649.311,E2 -1649.311} C_VEL
LIN {X 0,Y 580.295,Z 189.821,A -85,B 0,C 180,E1 -1652.201,E2 -1652.201} C_VEL
LIN {X 0,Y 580.295,Z 189.826,A -85,B 0,C 180,E1 -1654.696,E2 -1654.696} C_VEL
LIN {X 0,Y 580.295,Z 189.824,A -85,B 0,C 180,E1 -1657.269,E2 -1657.269} C_VEL
LIN {X 0,Y 580.293,Z 189.822,A -85,B 0,C 180,E1 -1660.272,E2 -1660.272} C_VEL
LIN {X 0,Y 580.272,Z 189.831,A -85,B 0,C 180,E1 -1662.707,E2 -1662.707} C_VEL
LIN {X 0,Y 580.27,Z 189.824,A -85,B 0,C 180,E1 -1665.609,E2 -1665.609} C_VEL
LIN {X 0,Y 580.31,Z 189.821,A -85,B 0,C 180,E1 -1668.235,E2 -1668.235} C_VEL
LIN {X 0,Y 580.28,Z 189.828,A -85,B 0,C 180,E1 -1670.966,E2 -1670.966} C_VEL
LIN {X 0,Y 580.265,Z 189.824,A -85,B 0,C 180,E1 -1673.597,E2 -1673.597} C_VEL
LIN {X 0,Y 580.314,Z 189.821,A -85,B 0,C 180,E1 -1676.146,E2 -1676.146} C_VEL
LIN {X 0,Y 580.281,Z 189.831,A -85,B 0,C 180,E1 -1678.616,E2 -1678.616} C_VEL
LIN {X 0,Y 580.292,Z 189.825,A -85,B 0,C 180,E1 -1681.025,E2 -1681.025} C_VEL
LIN {X 0,Y 580.291,Z 189.822,A -85,B 0,C 180,E1 -1683.667,E2 -1683.667} C_VEL
LIN {X 0,Y 580.299,Z 189.823,A -85,B 0,C 180,E1 -1685.684,E2 -1685.684} C_VEL
LIN {X 0,Y 580.309,Z 189.964,A -85,B 0,C 180,E1 -1686.95,E2 -1686.95} C_VEL
LIN {X 0,Y 580.987,Z 194.447,A -85,B 0,C 180,E1 -1687.602,E2 -1687.602} C_VEL
LIN {X 0,Y 580.802,Z 215.712,A -85,B 0,C 180,E1 -1690.52,E2 -1690.52} C_VEL
LIN {X 0,Y 580.749,Z 216.93,A -85,B 0,C 180,E1 -1690.684,E2 -1690.684} C_VEL
LIN {X 0,Y 581.874,Z 222.7,A -85,B 0,C 180,E1 -1690.798,E2 -1690.798} C_VEL
LIN {X 0,Y 581.528,Z 382.082,A -85,B 0,C 180,E1 -1692.835,E2 -1692.835} C_VEL
LIN {X 0,Y 581.41,Z 397.739,A -85,B 0,C 180,E1 -1693.181,E2 -1693.181} C_VEL
LIN {X 0,Y 581.227,Z 413.06,A -85,B 0,C 180,E1 -1693.673,E2 -1693.673} C_VEL
LIN {X 0,Y 581.117,Z 427.721,A -85,B 0,C 180,E1 -1694.3,E2 -1694.3} C_VEL
LIN {X 0,Y 580.927,Z 441.029,A -85,B 0,C 180,E1 -1695.014,E2 -1695.014} C_VEL
LIN {X 0,Y 580.791,Z 454.377,A -85,B 0,C 180,E1 -1695.89,E2 -1695.89} C_VEL
LIN {X 0,Y 580.592,Z 466.878,A -85,B 0,C 180,E1 -1696.882,E2 -1696.882} C_VEL
LIN {X 0,Y 580.46,Z 478.076,A -85,B 0,C 180,E1 -1697.945,E2 -1697.945} C_VEL
LIN {X 0,Y 580.337,Z 489.114,A -85,B 0,C 180,E1 -1699.201,E2 -1699.201} C_VEL
LIN {X 0,Y 580.239,Z 497.999,A -85,B 0,C 180,E1 -1700.413,E2 -1700.413} C_VEL
LIN {X 0,Y 580.195,Z 505.491,A -85,B 0,C 180,E1 -1701.642,E2 -1701.642} C_VEL
LIN {X 0,Y 580.139,Z 512.495,A -85,B 0,C 180,E1 -1703.042,E2 -1703.042} C_VEL
LIN {X 0,Y 580.127,Z 518.004,A -85,B 0,C 180,E1 -1704.438,E2 -1704.438} C_VEL
LIN {X 0,Y 580.087,Z 522.174,A -85,B 0,C 180,E1 -1705.831,E2 -1705.831} C_VEL
LIN {X 0,Y 580.038,Z 525.113,A -85,B 0,C 180,E1 -1707.222,E2 -1707.222} C_VEL
LIN {X 0,Y 580.043,Z 526.88,A -85,B 0,C 180,E1 -1708.611,E2 -1708.611} C_VEL
LIN {X 0,Y 580.035,Z 527.496,A -85,B 0,C 180,E1 -1710,E2 -1710} C_VEL
LIN {X 0,Y 580.045,Z 526.943,A -85,B 0,C 180,E1 -1711.389,E2 -1711.389} C_VEL
LIN {X 0,Y 580.04,Z 525.26,A -85,B 0,C 180,E1 -1712.778,E2 -1712.778} C_VEL
LIN {X 0,Y 580.087,Z 522.405,A -85,B 0,C 180,E1 -1714.169,E2 -1714.169} C_VEL
LIN {X 0,Y 580.123,Z 518.322,A -85,B 0,C 180,E1 -1715.562,E2 -1715.562} C_VEL
LIN {X 0,Y 580.139,Z 512.91,A -85,B 0,C 180,E1 -1716.958,E2 -1716.958} C_VEL
LIN {X 0,Y 580.19,Z 506.011,A -85,B 0,C 180,E1 -1718.358,E2 -1718.358} C_VEL
LIN {X 0,Y 580.235,Z 497.405,A -85,B 0,C 180,E1 -1719.763,E2 -1719.763} C_VEL
LIN {X 0,Y 580.308,Z 487.833,A -85,B 0,C 180,E1 -1721.046,E2 -1721.046} C_VEL
LIN {X 0,Y 580.472,Z 477.202,A -85,B 0,C 180,E1 -1722.232,E2 -1722.232} C_VEL
LIN {X 0,Y 580.606,Z 465.829,A -85,B 0,C 180,E1 -1723.296,E2 -1723.296} C_VEL
LIN {X 0,Y 580.759,Z 453.076,A -85,B 0,C 180,E1 -1724.291,E2 -1724.291} C_VEL
LIN {X 0,Y 580.931,Z 439.469,A -85,B 0,C 180,E1 -1725.166,E2 -1725.166} C_VEL
LIN {X 0,Y 581.115,Z 425.794,A -85,B 0,C 180,E1 -1725.88,E2 -1725.88} C_VEL
LIN {X 0,Y 581.275,Z 411.803,A -85,B 0,C 180,E1 -1726.461,E2 -1726.461} C_VEL
LIN {X 0,Y 581.455,Z 396.768,A -85,B 0,C 180,E1 -1726.932,E2 -1726.932} C_VEL
LIN {X 0,Y 581.528,Z 382.357,A -85,B 0,C 180,E1 -1727.25,E2 -1727.25} C_VEL
LIN {X 0,Y 581.807,Z 222.013,A -85,B 0,C 180,E1 -1729.303,E2 -1729.303} C_VEL
LIN {X 0,Y 580.782,Z 216.91,A -85,B 0,C 180,E1 -1729.408,E2 -1729.408} C_VEL
LIN {X 0,Y 580.973,Z 196.446,A -85,B 0,C 180,E1 -1732.211,E2 -1732.211} C_VEL
LIN {X 0,Y 580.819,Z 192.395,A -85,B 0,C 180,E1 -1732.78,E2 -1732.78} C_VEL
LIN {X 0,Y 580.288,Z 189.829,A -85,B 0,C 180,E1 -1733.166,E2 -1733.166} C_VEL
LIN {X 0,Y 580.294,Z 189.828,A -85,B 0,C 180,E1 -1735.848,E2 -1735.848} C_VEL
LIN {X 0,Y 580.299,Z 189.822,A -85,B 0,C 180,E1 -1738.185,E2 -1738.185} C_VEL
LIN {X 0,Y 580.283,Z 189.823,A -85,B 0,C 180,E1 -1740.694,E2 -1740.694} C_VEL
LIN {X 0,Y 580.304,Z 189.828,A -85,B 0,C 180,E1 -1743.316,E2 -1743.316} C_VEL
LIN {X 0,Y 580.261,Z 189.83,A -85,B 0,C 180,E1 -1745.758,E2 -1745.758} C_VEL
LIN {X 0,Y 580.285,Z 189.823,A -85,B 0,C 180,E1 -1748.145,E2 -1748.145} C_VEL
LIN {X 0,Y 580.296,Z 189.822,A -85,B 0,C 180,E1 -1750.842,E2 -1750.842} C_VEL
LIN {X 0,Y 580.284,Z 189.826,A -85,B 0,C 180,E1 -1753.656,E2 -1753.656} C_VEL
LIN {X 0,Y 580.271,Z 189.824,A -85,B 0,C 180,E1 -1756.609,E2 -1756.609} C_VEL
LIN {X 0,Y 580.294,Z 189.828,A -85,B 0,C 180,E1 -1759.156,E2 -1759.156} C_VEL
LIN {X 0,Y 580.285,Z 189.82,A -85,B 0,C 180,E1 -1761.926,E2 -1761.926} C_VEL
LIN {X 0,Y 580.302,Z 189.82,A -85,B 0,C 180,E1 -1764.456,E2 -1764.456} C_VEL
LIN {X 0,Y 580.284,Z 189.829,A -85,B 0,C 180,E1 -1766.975,E2 -1766.975} C_VEL
LIN {X 0,Y 580.303,Z 189.823,A -85,B 0,C 180,E1 -1769.425,E2 -1769.425} C_VEL
LIN {X 0,Y 580.312,Z 189.818,A -85,B 0,C 180,E1 -1772.136,E2 -1772.136} C_VEL
LIN {X 0,Y 580.313,Z 189.824,A -85,B 0,C 180,E1 -1775.269,E2 -1775.269} C_VEL
LIN {X 0,Y 580.266,Z 189.823,A -85,B 0,C 180,E1 -1777.947,E2 -1777.947} C_VEL
LIN {X 0,Y 580.309,Z 189.828,A -85,B 0,C 180,E1 -1780.914,E2 -1780.914} C_VEL
LIN {X 0,Y 580.276,Z 189.823,A -85,B 0,C 180,E1 -1783.825,E2 -1783.825} C_VEL
LIN {X 0,Y 580.274,Z 189.829,A -85,B 0,C 180,E1 -1786.696,E2 -1786.696} C_VEL
LIN {X 0,Y 580.295,Z 189.82,A -85,B 0,C 180,E1 -1789.533,E2 -1789.533} C_VEL
LIN {X 0,Y 580.323,Z 189.82,A -85,B 0,C 180,E1 -1792.344,E2 -1792.344} C_VEL
LIN {X 0,Y 580.334,Z 189.819,A -85,B 0,C 180,E1 -1795.137,E2 -1795.137} C_VEL
LIN {X 0,Y 580.325,Z 189.817,A -85,B 0,C 180,E1 -1797.918,E2 -1797.918} C_VEL
LIN {X 0,Y 580.36,Z 189.822,A -85,B 0,C 180,E1 -1800.694,E2 -1800.694} C_VEL
LIN {X 0,Y 580.281,Z 189.821,A -85,B 0,C 180,E1 -1803.472,E2 -1803.472} C_VEL
LIN {X 0,Y 580.318,Z 189.817,A -85,B 0,C 180,E1 -1805.56,E2 -1805.56} C_VEL
LIN {X 0,Y 580.326,Z 189.823,A -85,B 0,C 180,E1 -1808.356,E2 -1808.356} C_VEL
LIN {X 0,Y 580.323,Z 189.818,A -85,B 0,C 180,E1 -1811.208,E2 -1811.208} C_VEL
LIN {X 0,Y 580.305,Z 189.827,A -85,B 0,C 180,E1 -1814.339,E2 -1814.339} C_VEL
LIN {X 0,Y 580.306,Z 189.821,A -85,B 0,C 180,E1 -1816.916,E2 -1816.916} C_VEL
LIN {X 0,Y 580.299,Z 189.822,A -85,B 0,C 180,E1 -1819.822,E2 -1819.822} C_VEL
LIN {X 0,Y 580.267,Z 189.828,A -85,B 0,C 180,E1 -1822.053,E2 -1822.053} C_VEL
LIN {X 0,Y 580.297,Z 189.82,A -85,B 0,C 180,E1 -1825.08,E2 -1825.08} C_VEL
LIN {X 0,Y 580.294,Z 189.83,A -85,B 0,C 180,E1 -1828.186,E2 -1828.186} C_VEL
LIN {X 0,Y 580.291,Z 189.824,A -85,B 0,C 180,E1 -1830.698,E2 -1830.698} C_VEL
LIN {X 0,Y 580.295,Z 189.82,A -85,B 0,C 180,E1 -1833.317,E2 -1833.317} C_VEL
LIN {X 0,Y 580.318,Z 189.821,A -85,B 0,C 180,E1 -1835.768,E2 -1835.768} C_VEL
LIN {X 0,Y 580.283,Z 189.831,A -85,B 0,C 180,E1 -1838.147,E2 -1838.147} C_VEL
LIN {X 0,Y 580.296,Z 189.819,A -85,B 0,C 180,E1 -1840.844,E2 -1840.844} C_VEL
LIN {X 0,Y 580.273,Z 189.827,A -85,B 0,C 180,E1 -1843.658,E2 -1843.658} C_VEL
LIN {X 0,Y 580.279,Z 189.824,A -85,B 0,C 180,E1 -1846.609,E2 -1846.609} C_VEL
LIN {X 0,Y 580.295,Z 189.821,A -85,B 0,C 180,E1 -1849.157,E2 -1849.157} C_VEL
LIN {X 0,Y 580.286,Z 189.83,A -85,B 0,C 180,E1 -1851.928,E2 -1851.928} C_VEL
LIN {X 0,Y 580.281,Z 189.825,A -85,B 0,C 180,E1 -1854.456,E2 -1854.456} C_VEL
LIN {X 0,Y 580.288,Z 189.822,A -85,B 0,C 180,E1 -1856.976,E2 -1856.976} C_VEL
LIN {X 0,Y 580.292,Z 189.825,A -85,B 0,C 180,E1 -1859.426,E2 -1859.426} C_VEL
LIN {X 0,Y 580.288,Z 189.829,A -85,B 0,C 180,E1 -1862.143,E2 -1862.143} C_VEL
LIN {X 0,Y 580.363,Z 190.012,A -85,B 0,C 180,E1 -1863.893,E2 -1863.893} C_VEL
LIN {X 0,Y 581.423,Z 195.344,A -85,B 0,C 180,E1 -1864.59,E2 -1864.59} C_VEL
LIN {X 0,Y 581.201,Z 217.275,A -85,B 0,C 180,E1 -1867.236,E2 -1867.236} C_VEL
LIN {X 0,Y 580.959,Z 242.245,A -85,B 0,C 180,E1 -1870.201,E2 -1870.201} C_VEL
LIN {X 0,Y 580.896,Z 245.908,A -85,B 0,C 180,E1 -1870.631,E2 -1870.631} C_VEL
LIN {X 0,Y 581.9,Z 251.764,A -85,B 0,C 180,E1 -1870.742,E2 -1870.742} C_VEL
LIN {X 0,Y 581.529,Z 412.49,A -85,B 0,C 180,E1 -1872.798,E2 -1872.798} C_VEL
LIN {X 0,Y 581.412,Z 427.721,A -85,B 0,C 180,E1 -1873.136,E2 -1873.136} C_VEL
LIN {X 0,Y 581.256,Z 443.052,A -85,B 0,C 180,E1 -1873.628,E2 -1873.628} C_VEL
LIN {X 0,Y 581.123,Z 456.778,A -85,B 0,C 180,E1 -1874.21,E2 -1874.21} C_VEL
LIN {X 0,Y 580.95,Z 470.249,A -85,B 0,C 180,E1 -1874.925,E2 -1874.925} C_VEL
LIN {X 0,Y 580.804,Z 483.485,A -85,B 0,C 180,E1 -1875.784,E2 -1875.784} C_VEL
LIN {X 0,Y 580.608,Z 495.293,A -85,B 0,C 180,E1 -1876.704,E2 -1876.704} C_VEL
LIN {X 0,Y 580.478,Z 506.752,A -85,B 0,C 180,E1 -1877.768,E2 -1877.768} C_VEL
LIN {X 0,Y 580.308,Z 517.453,A -85,B 0,C 180,E1 -1878.953,E2 -1878.953} C_VEL
LIN {X 0,Y 580.268,Z 525.859,A -85,B 0,C 180,E1 -1880.062,E2 -1880.062} C_VEL
LIN {X 0,Y 580.215,Z 533.734,A -85,B 0,C 180,E1 -1881.292,E2 -1881.292} C_VEL
LIN {X 0,Y 580.13,Z 541.09,A -85,B 0,C 180,E1 -1882.692,E2 -1882.692} C_VEL
LIN {X 0,Y 580.132,Z 546.924,A -85,B 0,C 180,E1 -1884.09,E2 -1884.09} C_VEL
LIN {X 0,Y 580.041,Z 550.385,A -85,B 0,C 180,E1 -1885.135,E2 -1885.135} C_VEL
LIN {X 0,Y 580.104,Z 553.889,A -85,B 0,C 180,E1 -1886.527,E2 -1886.527} C_VEL
LIN {X 0,Y 580.039,Z 556.193,A -85,B 0,C 180,E1 -1887.917,E2 -1887.917} C_VEL
LIN {X 0,Y 580.038,Z 557.349,A -85,B 0,C 180,E1 -1889.306,E2 -1889.306} C_VEL
LIN {X 0,Y 580.038,Z 557.349,A -85,B 0,C 180,E1 -1890.694,E2 -1890.694} C_VEL
LIN {X 0,Y 580.039,Z 556.191,A -85,B 0,C 180,E1 -1892.083,E2 -1892.083} C_VEL
LIN {X 0,Y 580.104,Z 553.887,A -85,B 0,C 180,E1 -1893.473,E2 -1893.473} C_VEL
LIN {X 0,Y 580.041,Z 550.385,A -85,B 0,C 180,E1 -1894.865,E2 -1894.865} C_VEL
LIN {X 0,Y 580.093,Z 545.609,A -85,B 0,C 180,E1 -1896.26,E2 -1896.26} C_VEL
LIN {X 0,Y 580.165,Z 539.424,A -85,B 0,C 180,E1 -1897.657,E2 -1897.657} C_VEL
LIN {X 0,Y 580.207,Z 531.65,A -85,B 0,C 180,E1 -1899.06,E2 -1899.06} C_VEL
LIN {X 0,Y 580.308,Z 523.371,A -85,B 0,C 180,E1 -1900.29,E2 -1900.29} C_VEL
LIN {X 0,Y 580.382,Z 513.397,A -85,B 0,C 180,E1 -1901.525,E2 -1901.525} C_VEL
LIN {X 0,Y 580.541,Z 503.192,A -85,B 0,C 180,E1 -1902.586,E2 -1902.586} C_VEL
LIN {X 0,Y 580.677,Z 491.023,A -85,B 0,C 180,E1 -1903.651,E2 -1903.651} C_VEL
LIN {X 0,Y 580.874,Z 477.533,A -85,B 0,C 180,E1 -1904.625,E2 -1904.625} C_VEL
LIN {X 0,Y 581.045,Z 463.876,A -85,B 0,C 180,E1 -1905.432,E2 -1905.432} C_VEL
LIN {X 0,Y 581.214,Z 449.807,A -85,B 0,C 180,E1 -1906.102,E2 -1906.102} C_VEL
LIN {X 0,Y 581.356,Z 435.315,A -85,B 0,C 180,E1 -1906.64,E2 -1906.64} C_VEL
LIN {X 0,Y 581.486,Z 420.069,A -85,B 0,C 180,E1 -1907.052,E2 -1907.052} C_VEL
LIN {X 0,Y 581.551,Z 404.554,A -85,B 0,C 180,E1 -1907.323,E2 -1907.323} C_VEL
LIN {X 0,Y 581.801,Z 250.662,A -85,B 0,C 180,E1 -1909.276,E2 -1909.276} C_VEL
LIN {X 0,Y 580.899,Z 245.763,A -85,B 0,C 180,E1 -1909.386,E2 -1909.386} C_VEL
LIN {X 0,Y 581.197,Z 220.396,A -85,B 0,C 180,E1 -1912.389,E2 -1912.389} C_VEL
LIN {X 0,Y 581.431,Z 198.501,A -85,B 0,C 180,E1 -1915.027,E2 -1915.027} C_VEL
LIN {X 0,Y 581.215,Z 193.758,A -85,B 0,C 180,E1 -1915.612,E2 -1915.612} C_VEL
LIN {X 0,Y 580.315,Z 189.828,A -85,B 0,C 180,E1 -1916.147,E2 -1916.147} C_VEL
LIN {X 0,Y 580.288,Z 189.823,A -85,B 0,C 180,E1 -1918.976,E2 -1918.976} C_VEL
LIN {X 0,Y 580.272,Z 189.823,A -85,B 0,C 180,E1 -1921.385,E2 -1921.385} C_VEL
LIN {X 0,Y 580.313,Z 189.822,A -85,B 0,C 180,E1 -1923.854,E2 -1923.854} C_VEL
LIN {X 0,Y 580.297,Z 189.821,A -85,B 0,C 180,E1 -1926.934,E2 -1926.934} C_VEL
LIN {X 0,Y 580.289,Z 189.83,A -85,B 0,C 180,E1 -1929.932,E2 -1929.932} C_VEL
LIN {X 0,Y 580.275,Z 189.824,A -85,B 0,C 180,E1 -1932.705,E2 -1932.705} C_VEL
LIN {X 0,Y 580.264,Z 189.828,A -85,B 0,C 180,E1 -1935.608,E2 -1935.608} C_VEL
LIN {X 0,Y 580.308,Z 189.824,A -85,B 0,C 180,E1 -1938.234,E2 -1938.234} C_VEL
LIN {X 0,Y 580.284,Z 189.821,A -85,B 0,C 180,E1 -1940.966,E2 -1940.966} C_VEL
LIN {X 0,Y 580.29,Z 189.826,A -85,B 0,C 180,E1 -1943.598,E2 -1943.598} C_VEL
LIN {X 0,Y 580.312,Z 189.822,A -85,B 0,C 180,E1 -1946.145,E2 -1946.145} C_VEL
LIN {X 0,Y 580.282,Z 189.822,A -85,B 0,C 180,E1 -1948.615,E2 -1948.615} C_VEL
LIN {X 0,Y 580.286,Z 189.821,A -85,B 0,C 180,E1 -1951.024,E2 -1951.024} C_VEL
LIN {X 0,Y 580.283,Z 189.831,A -85,B 0,C 180,E1 -1953.665,E2 -1953.665} C_VEL
LIN {X 0,Y 580.292,Z 189.831,A -85,B 0,C 180,E1 -1955.683,E2 -1955.683} C_VEL
LIN {X 0,Y 580.267,Z 189.827,A -85,B 0,C 180,E1 -1957.947,E2 -1957.947} C_VEL
LIN {X 0,Y 580.309,Z 189.819,A -85,B 0,C 180,E1 -1960.914,E2 -1960.914} C_VEL
LIN {X 0,Y 580.275,Z 189.829,A -85,B 0,C 180,E1 -1963.826,E2 -1963.826} C_VEL
LIN {X 0,Y 580.273,Z 189.823,A -85,B 0,C 180,E1 -1966.696,E2 -1966.696} C_VEL
LIN {X 0,Y 580.295,Z 189.83,A -85,B 0,C 180,E1 -1969.533,E2 -1969.533} C_VEL
LIN {X 0,Y 580.324,Z 189.816,A -85,B 0,C 180,E1 -1972.345,E2 -1972.345} C_VEL
LIN {X 0,Y 580.338,Z 189.82,A -85,B 0,C 180,E1 -1975.137,E2 -1975.137} C_VEL
LIN {X 0,Y 580.327,Z 189.819,A -85,B 0,C 180,E1 -1977.918,E2 -1977.918} C_VEL
LIN {X 0,Y 580.359,Z 189.813,A -85,B 0,C 180,E1 -1980.694,E2 -1980.694} C_VEL
LIN {X 0,Y 580.282,Z 189.829,A -85,B 0,C 180,E1 -1983.472,E2 -1983.472} C_VEL
LIN {X 0,Y 580.321,Z 189.823,A -85,B 0,C 180,E1 -1985.56,E2 -1985.56} C_VEL
LIN {X 0,Y 580.327,Z 189.816,A -85,B 0,C 180,E1 -1988.356,E2 -1988.356} C_VEL
LIN {X 0,Y 580.324,Z 189.827,A -85,B 0,C 180,E1 -1991.209,E2 -1991.209} C_VEL
LIN {X 0,Y 580.306,Z 189.819,A -85,B 0,C 180,E1 -1994.339,E2 -1994.339} C_VEL
LIN {X 0,Y 580.305,Z 189.825,A -85,B 0,C 180,E1 -1996.915,E2 -1996.915} C_VEL
LIN {X 0,Y 580.299,Z 189.82,A -85,B 0,C 180,E1 -1999.823,E2 -1999.823} C_VEL
LIN {X 0,Y 580.273,Z 189.829,A -85,B 0,C 180,E1 -2001.342,E2 -2001.342} C_VEL
LIN {X 0,Y 579.578,Z 189.912,A -85,B 0,C 180,E1 -2001.921,E2 -2001.921} C_VEL
LIN {X 0,Y 576.703,Z 190.274,A -85,B 0,C 180,E1 -2002.861,E2 -2002.861} C_VEL
LIN {X 0,Y 574.309,Z 190.568,A -85,B 0,C 180,E1 -2003.618,E2 -2003.618} C_VEL
LIN {X 0,Y 573.31,Z 190.69,A -85,B 0,C 180,E1 -2004.201,E2 -2004.201} C_VEL
LIN {X 0,Y 573.243,Z 190.699,A -85,B 0,C 180,E1 -2004.399,E2 -2004.399} C_VEL
LIN {X 0,Y 573.247,Z 190.704,A -85,B 0,C 180,E1 -2006.976,E2 -2006.976} C_VEL
LIN {X 0,Y 573.245,Z 190.701,A -85,B 0,C 180,E1 -2009.49,E2 -2009.49} C_VEL
LIN {X 0,Y 573.248,Z 190.699,A -85,B 0,C 180,E1 -2012.23,E2 -2012.23} C_VEL
LIN {X 0,Y 573.246,Z 190.705,A -85,B 0,C 180,E1 -2014.775,E2 -2014.775} C_VEL
LIN {X 0,Y 573.248,Z 190.703,A -85,B 0,C 180,E1 -2017.167,E2 -2017.167} C_VEL
LIN {X 0,Y 573.243,Z 190.699,A -85,B 0,C 180,E1 -2019.608,E2 -2019.608} C_VEL
LIN {X 0,Y 573.235,Z 190.706,A -85,B 0,C 180,E1 -2022.642,E2 -2022.642} C_VEL
LIN {X 0,Y 573.235,Z 190.7,A -85,B 0,C 180,E1 -2025.668,E2 -2025.668} C_VEL
LIN {X 0,Y 573.241,Z 190.706,A -85,B 0,C 180,E1 -2028.545,E2 -2028.545} C_VEL
LIN {X 0,Y 573.242,Z 190.701,A -85,B 0,C 180,E1 -2031.299,E2 -2031.299} C_VEL
LIN {X 0,Y 573.21,Z 190.704,A -85,B 0,C 180,E1 -2034.019,E2 -2034.019} C_VEL
LIN {X 0,Y 573.284,Z 190.703,A -85,B 0,C 180,E1 -2036.52,E2 -2036.52} C_VEL
LIN {X 0,Y 573.231,Z 190.704,A -85,B 0,C 180,E1 -2039.118,E2 -2039.118} C_VEL
LIN {X 0,Y 573.251,Z 190.701,A -85,B 0,C 180,E1 -2041.972,E2 -2041.972} C_VEL
LIN {X 0,Y 573.254,Z 190.707,A -85,B 0,C 180,E1 -2044.591,E2 -2044.591} C_VEL
LIN {X 0,Y 573.264,Z 190.799,A -85,B 0,C 180,E1 -2046.752,E2 -2046.752} C_VEL
LIN {X 0,Y 574.097,Z 195.828,A -85,B 0,C 180,E1 -2047.508,E2 -2047.508} C_VEL
LIN {X 0,Y 573.854,Z 216.921,A -85,B 0,C 180,E1 -2050.44,E2 -2050.44} C_VEL
LIN {X 0,Y 575.181,Z 223.44,A -85,B 0,C 180,E1 -2050.575,E2 -2050.575} C_VEL
LIN {X 0,Y 574.741,Z 382.222,A -85,B 0,C 180,E1 -2052.628,E2 -2052.628} C_VEL
LIN {X 0,Y 574.615,Z 397.759,A -85,B 0,C 180,E1 -2052.976,E2 -2052.976} C_VEL
LIN {X 0,Y 574.423,Z 413.073,A -85,B 0,C 180,E1 -2053.474,E2 -2053.474} C_VEL
LIN {X 0,Y 574.252,Z 427.73,A -85,B 0,C 180,E1 -2054.108,E2 -2054.108} C_VEL
LIN {X 0,Y 574.037,Z 441.041,A -85,B 0,C 180,E1 -2054.83,E2 -2054.83} C_VEL
LIN {X 0,Y 573.858,Z 454.559,A -85,B 0,C 180,E1 -2055.729,E2 -2055.729} C_VEL
LIN {X 0,Y 573.631,Z 466.885,A -85,B 0,C 180,E1 -2056.72,E2 -2056.72} C_VEL
LIN {X 0,Y 573.458,Z 478.082,A -85,B 0,C 180,E1 -2057.795,E2 -2057.795} C_VEL
LIN {X 0,Y 573.294,Z 487.583,A -85,B 0,C 180,E1 -2058.877,E2 -2058.877} C_VEL
LIN {X 0,Y 573.203,Z 496.777,A -85,B 0,C 180,E1 -2060.116,E2 -2060.116} C_VEL
LIN {X 0,Y 573.134,Z 504.486,A -85,B 0,C 180,E1 -2061.361,E2 -2061.361} C_VEL
LIN {X 0,Y 573.075,Z 510.883,A -85,B 0,C 180,E1 -2062.602,E2 -2062.602} C_VEL
LIN {X 0,Y 573.042,Z 516.767,A -85,B 0,C 180,E1 -2064.016,E2 -2064.016} C_VEL
LIN {X 0,Y 572.949,Z 520.251,A -85,B 0,C 180,E1 -2065.074,E2 -2065.074} C_VEL
LIN {X 0,Y 573.004,Z 523.795,A -85,B 0,C 180,E1 -2066.484,E2 -2066.484} C_VEL
LIN {X 0,Y 572.938,Z 526.139,A -85,B 0,C 180,E1 -2067.891,E2 -2067.891} C_VEL
LIN {X 0,Y 572.936,Z 527.337,A -85,B 0,C 180,E1 -2069.297,E2 -2069.297} C_VEL
LIN {X 0,Y 572.937,Z 527.359,A -85,B 0,C 180,E1 -2070.703,E2 -2070.703} C_VEL
LIN {X 0,Y 572.939,Z 526.243,A -85,B 0,C 180,E1 -2072.109,E2 -2072.109} C_VEL
LIN {X 0,Y 573.006,Z 523.981,A -85,B 0,C 180,E1 -2073.516,E2 -2073.516} C_VEL
LIN {X 0,Y 572.949,Z 520.521,A -85,B 0,C 180,E1 -2074.926,E2 -2074.926} C_VEL
LIN {X 0,Y 573.007,Z 515.788,A -85,B 0,C 180,E1 -2076.337,E2 -2076.337} C_VEL
LIN {X 0,Y 573.094,Z 509.655,A -85,B 0,C 180,E1 -2077.752,E2 -2077.752} C_VEL
LIN {X 0,Y 573.134,Z 501.934,A -85,B 0,C 180,E1 -2079.172,E2 -2079.172} C_VEL
LIN {X 0,Y 573.265,Z 493.696,A -85,B 0,C 180,E1 -2080.418,E2 -2080.418} C_VEL
LIN {X 0,Y 573.354,Z 483.787,A -85,B 0,C 180,E1 -2081.668,E2 -2081.668} C_VEL
LIN {X 0,Y 573.534,Z 473.636,A -85,B 0,C 180,E1 -2082.742,E2 -2082.742} C_VEL
LIN {X 0,Y 573.721,Z 461.557,A -85,B 0,C 180,E1 -2083.82,E2 -2083.82} C_VEL
LIN {X 0,Y 573.919,Z 448.602,A -85,B 0,C 180,E1 -2084.78,E2 -2084.78} C_VEL
LIN {X 0,Y 574.141,Z 434.722,A -85,B 0,C 180,E1 -2085.622,E2 -2085.622} C_VEL
LIN {X 0,Y 574.346,Z 419.793,A -85,B 0,C 180,E1 -2086.346,E2 -2086.346} C_VEL
LIN {X 0,Y 574.528,Z 405.281,A -85,B 0,C 180,E1 -2086.889,E2 -2086.889} C_VEL
LIN {X 0,Y 574.685,Z 389.714,A -85,B 0,C 180,E1 -2087.313,E2 -2087.313} C_VEL
LIN {X 0,Y 574.771,Z 373.498,A -85,B 0,C 180,E1 -2087.593,E2 -2087.593} C_VEL
LIN {X 0,Y 575.103,Z 222.959,A -85,B 0,C 180,E1 -2089.524,E2 -2089.524} C_VEL
LIN {X 0,Y 573.832,Z 216.88,A -85,B 0,C 180,E1 -2089.656,E2 -2089.656} C_VEL
LIN {X 0,Y 574.09,Z 197.797,A -85,B 0,C 180,E1 -2092.302,E2 -2092.302} C_VEL
LIN {X 0,Y 573.892,Z 193.806,A -85,B 0,C 180,E1 -2092.88,E2 -2092.88} C_VEL
LIN {X 0,Y 573.251,Z 190.707,A -85,B 0,C 180,E1 -2093.375,E2 -2093.375} C_VEL
LIN {X 0,Y 573.264,Z 190.7,A -85,B 0,C 180,E1 -2096.189,E2 -2096.189} C_VEL
LIN {X 0,Y 573.237,Z 190.701,A -85,B 0,C 180,E1 -2098.564,E2 -2098.564} C_VEL
LIN {X 0,Y 573.227,Z 190.704,A -85,B 0,C 180,E1 -2100.992,E2 -2100.992} C_VEL
LIN {X 0,Y 573.26,Z 190.706,A -85,B 0,C 180,E1 -2103.523,E2 -2103.523} C_VEL
LIN {X 0,Y 573.236,Z 190.701,A -85,B 0,C 180,E1 -2106.049,E2 -2106.049} C_VEL
LIN {X 0,Y 573.244,Z 190.701,A -85,B 0,C 180,E1 -2108.7,E2 -2108.7} C_VEL
LIN {X 0,Y 573.25,Z 190.704,A -85,B 0,C 180,E1 -2111.595,E2 -2111.595} C_VEL
LIN {X 0,Y 573.235,Z 190.7,A -85,B 0,C 180,E1 -2114.332,E2 -2114.332} C_VEL
LIN {X 0,Y 573.235,Z 190.707,A -85,B 0,C 180,E1 -2117.358,E2 -2117.358} C_VEL
LIN {X 0,Y 573.243,Z 190.699,A -85,B 0,C 180,E1 -2120.392,E2 -2120.392} C_VEL
LIN {X 0,Y 573.25,Z 190.704,A -85,B 0,C 180,E1 -2123.077,E2 -2123.077} C_VEL
LIN {X 0,Y 573.268,Z 190.698,A -85,B 0,C 180,E1 -2125.671,E2 -2125.671} C_VEL
LIN {X 0,Y 573.242,Z 190.696,A -85,B 0,C 180,E1 -2128.185,E2 -2128.185} C_VEL
LIN {X 0,Y 573.261,Z 190.699,A -85,B 0,C 180,E1 -2130.634,E2 -2130.634} C_VEL
LIN {X 0,Y 573.243,Z 190.708,A -85,B 0,C 180,E1 -2133.024,E2 -2133.024} C_VEL
LIN {X 0,Y 573.267,Z 190.7,A -85,B 0,C 180,E1 -2135.366,E2 -2135.366} C_VEL
LIN {X 0,Y 573.223,Z 190.703,A -85,B 0,C 180,E1 -2138.419,E2 -2138.419} C_VEL
LIN {X 0,Y 573.271,Z 190.702,A -85,B 0,C 180,E1 -2140.727,E2 -2140.727} C_VEL
LIN {X 0,Y 573.251,Z 190.699,A -85,B 0,C 180,E1 -2143.622,E2 -2143.622} C_VEL
LIN {X 0,Y 573.231,Z 190.704,A -85,B 0,C 180,E1 -2146.529,E2 -2146.529} C_VEL
LIN {X 0,Y 573.273,Z 190.704,A -85,B 0,C 180,E1 -2148.734,E2 -2148.734} C_VEL
LIN {X 0,Y 573.282,Z 190.694,A -85,B 0,C 180,E1 -2151.54,E2 -2151.54} C_VEL
LIN {X 0,Y 573.287,Z 190.697,A -85,B 0,C 180,E1 -2154.372,E2 -2154.372} C_VEL
LIN {X 0,Y 573.297,Z 190.692,A -85,B 0,C 180,E1 -2157.892,E2 -2157.892} C_VEL
LIN {X 0,Y 573.33,Z 190.697,A -85,B 0,C 180,E1 -2160.702,E2 -2160.702} C_VEL
LIN {X 0,Y 573.233,Z 190.699,A -85,B 0,C 180,E1 -2163.514,E2 -2163.514} C_VEL
LIN {X 0,Y 573.284,Z 190.694,A -85,B 0,C 180,E1 -2165.628,E2 -2165.628} C_VEL
LIN {X 0,Y 573.298,Z 190.7,A -85,B 0,C 180,E1 -2168.459,E2 -2168.459} C_VEL
LIN {X 0,Y 573.289,Z 190.694,A -85,B 0,C 180,E1 -2171.312,E2 -2171.312} C_VEL
LIN {X 0,Y 573.271,Z 190.704,A -85,B 0,C 180,E1 -2174.425,E2 -2174.425} C_VEL
LIN {X 0,Y 573.251,Z 190.698,A -85,B 0,C 180,E1 -2177.112,E2 -2177.112} C_VEL
LIN {X 0,Y 573.248,Z 190.704,A -85,B 0,C 180,E1 -2180.077,E2 -2180.077} C_VEL
LIN {X 0,Y 573.231,Z 190.71,A -85,B 0,C 180,E1 -2182.338,E2 -2182.338} C_VEL
LIN {X 0,Y 573.245,Z 190.698,A -85,B 0,C 180,E1 -2185.41,E2 -2185.41} C_VEL
LIN {X 0,Y 573.256,Z 190.704,A -85,B 0,C 180,E1 -2188.032,E2 -2188.032} C_VEL
LIN {X 0,Y 573.236,Z 190.701,A -85,B 0,C 180,E1 -2190.885,E2 -2190.885} C_VEL
LIN {X 0,Y 573.254,Z 190.698,A -85,B 0,C 180,E1 -2193.525,E2 -2193.525} C_VEL
LIN {X 0,Y 573.254,Z 190.706,A -85,B 0,C 180,E1 -2196.049,E2 -2196.049} C_VEL
LIN {X 0,Y 573.237,Z 190.701,A -85,B 0,C 180,E1 -2198.702,E2 -2198.702} C_VEL
LIN {X 0,Y 573.247,Z 190.699,A -85,B 0,C 180,E1 -2201.596,E2 -2201.596} C_VEL
LIN {X 0,Y 573.229,Z 190.706,A -85,B 0,C 180,E1 -2204.334,E2 -2204.334} C_VEL
LIN {X 0,Y 573.237,Z 190.701,A -85,B 0,C 180,E1 -2207.359,E2 -2207.359} C_VEL
LIN {X 0,Y 573.242,Z 190.702,A -85,B 0,C 180,E1 -2210.394,E2 -2210.394} C_VEL
LIN {X 0,Y 573.251,Z 190.698,A -85,B 0,C 180,E1 -2213.078,E2 -2213.078} C_VEL
LIN {X 0,Y 573.263,Z 190.704,A -85,B 0,C 180,E1 -2215.672,E2 -2215.672} C_VEL
LIN {X 0,Y 573.237,Z 190.705,A -85,B 0,C 180,E1 -2218.185,E2 -2218.185} C_VEL
LIN {X 0,Y 573.262,Z 190.699,A -85,B 0,C 180,E1 -2220.635,E2 -2220.635} C_VEL
LIN {X 0,Y 573.262,Z 190.707,A -85,B 0,C 180,E1 -2223.62,E2 -2223.62} C_VEL
LIN {X 0,Y 574.565,Z 196.75,A -85,B 0,C 180,E1 -2224.459,E2 -2224.459} C_VEL
LIN {X 0,Y 574.398,Z 217.267,A -85,B 0,C 180,E1 -2226.951,E2 -2226.951} C_VEL
LIN {X 0,Y 574.051,Z 242.245,A -85,B 0,C 180,E1 -2229.953,E2 -2229.953} C_VEL
LIN {X 0,Y 574.057,Z 246.193,A -85,B 0,C 180,E1 -2230.396,E2 -2230.396} C_VEL
LIN {X 0,Y 575.214,Z 252.47,A -85,B 0,C 180,E1 -2230.518,E2 -2230.518} C_VEL
LIN {X 0,Y 574.763,Z 412.022,A -85,B 0,C 180,E1 -2232.58,E2 -2232.58} C_VEL
LIN {X 0,Y 574.626,Z 427.719,A -85,B 0,C 180,E1 -2232.931,E2 -2232.931} C_VEL
LIN {X 0,Y 574.437,Z 443.049,A -85,B 0,C 180,E1 -2233.428,E2 -2233.428} C_VEL
LIN {X 0,Y 574.264,Z 456.781,A -85,B 0,C 180,E1 -2234.017,E2 -2234.017} C_VEL
LIN {X 0,Y 574.036,Z 470.252,A -85,B 0,C 180,E1 -2234.739,E2 -2234.739} C_VEL
LIN {X 0,Y 573.86,Z 483.824,A -85,B 0,C 180,E1 -2235.632,E2 -2235.632} C_VEL
LIN {X 0,Y 573.635,Z 496.354,A -85,B 0,C 180,E1 -2236.63,E2 -2236.63} C_VEL
LIN {X 0,Y 573.477,Z 506.752,A -85,B 0,C 180,E1 -2237.616,E2 -2237.616} C_VEL
LIN {X 0,Y 573.286,Z 516.771,A -85,B 0,C 180,E1 -2238.734,E2 -2238.734} C_VEL
LIN {X 0,Y 573.243,Z 525.859,A -85,B 0,C 180,E1 -2239.939,E2 -2239.939} C_VEL
LIN {X 0,Y 573.133,Z 533.735,A -85,B 0,C 180,E1 -2241.183,E2 -2241.183} C_VEL
LIN {X 0,Y 573.074,Z 541.09,A -85,B 0,C 180,E1 -2242.602,E2 -2242.602} C_VEL
LIN {X 0,Y 573.042,Z 546.923,A -85,B 0,C 180,E1 -2244.016,E2 -2244.016} C_VEL
LIN {X 0,Y 572.951,Z 550.386,A -85,B 0,C 180,E1 -2245.074,E2 -2245.074} C_VEL
LIN {X 0,Y 573.004,Z 553.89,A -85,B 0,C 180,E1 -2246.484,E2 -2246.484} C_VEL
LIN {X 0,Y 572.938,Z 556.192,A -85,B 0,C 180,E1 -2247.891,E2 -2247.891} C_VEL
LIN {X 0,Y 572.938,Z 557.349,A -85,B 0,C 180,E1 -2249.297,E2 -2249.297} C_VEL
LIN {X 0,Y 572.938,Z 557.349,A -85,B 0,C 180,E1 -2250.703,E2 -2250.703} C_VEL
LIN {X 0,Y 572.938,Z 556.19,A -85,B 0,C 180,E1 -2252.109,E2 -2252.109} C_VEL
LIN {X 0,Y 573.004,Z 553.887,A -85,B 0,C 180,E1 -2253.516,E2 -2253.516} C_VEL
LIN {X 0,Y 572.951,Z 550.386,A -85,B 0,C 180,E1 -2254.926,E2 -2254.926} C_VEL
LIN {X 0,Y 573.014,Z 545.609,A -85,B 0,C 180,E1 -2256.337,E2 -2256.337} C_VEL
LIN {X 0,Y 573.093,Z 539.423,A -85,B 0,C 180,E1 -2257.752,E2 -2257.752} C_VEL
LIN {X 0,Y 573.135,Z 531.649,A -85,B 0,C 180,E1 -2259.172,E2 -2259.172} C_VEL
LIN {X 0,Y 573.27,Z 523.37,A -85,B 0,C 180,E1 -2260.418,E2 -2260.418} C_VEL
LIN {X 0,Y 573.385,Z 513.394,A -85,B 0,C 180,E1 -2261.668,E2 -2261.668} C_VEL
LIN {X 0,Y 573.567,Z 503.191,A -85,B 0,C 180,E1 -2262.741,E2 -2262.741} C_VEL
LIN {X 0,Y 573.742,Z 491.023,A -85,B 0,C 180,E1 -2263.819,E2 -2263.819} C_VEL
LIN {X 0,Y 573.962,Z 477.909,A -85,B 0,C 180,E1 -2264.781,E2 -2264.781} C_VEL
LIN {X 0,Y 574.146,Z 465.519,A -85,B 0,C 180,E1 -2265.531,E2 -2265.531} C_VEL
